arrEn[1] := bEn01;
arrEn[2] := bEn02;
arrEn[3] := bEn03;
arrEn[4] := bEn04;

arrVal[1] := bVal01;
arrVal[2] := bVal02;
arrVal[3] := bVal03;
arrVal[4] := bVal04;

bQ := FALSE;
bVal := FALSE;
nActvPrio := Const.nNoActvPrio;

FOR i := 1 TO cBA_PrioSwiB04 BY 1 DO
	IF	arrEn[i] = TRUE
	THEN
		bQ := TRUE;
		bVal := arrVal[i];
		nActvPrio := i;
		EXIT;
	END_IF
END_FOR

END_FUNCTION_BLOCK

// TEST/TestPackage/TEMPLATES/HeatSupply/HeatingCircuit/FB_Bnet_H_HtgCir_Sp
FUNCTION_BLOCK FB_Bnet_H_HtgCir_Sp EXTENDS FB_BACnet_View
VAR_INPUT
	rWthT			: REAL;
	nOpMod		: UDINT;	// Betriebsart	// Operating mode 
END_VAR
VAR_INPUT CONSTANT PERSISTENT
	HeatingSetpointProtection : REAL := 5;
END_VAR
VAR_OUTPUT
	rVal			: REAL;	//Sollwert Heizkreis//Setpoint heating circuit	
END_VAR
VAR_INPUT CONSTANT
	Curve							:	FB_Bnet_Scale_04 := (
											iParent			:= THIS^);
										
	NightOffs						:	FB_BACnet_AV_Setp := (
											iParent 			:= THIS^,
											sObjectName			:= '\/SP01',
											sDescription		:= '\/Sollwert Nachtabsenkung',
											eUnit				:= E_BA_Unit.eTemperature_DegreesCelsius,
											fValue				:= 8.0);

	SpFlWT							:	FB_BACnet_AV_Disp := (
											iParent 			:= THIS^,
											sObjectName			:= '\/SWC01',
											sDescription		:= '\/Errechnete Vorlauftemperatur',
											eUnit				:= E_BA_Unit.eTemperature_DegreesCelsius);
END_VAR
VAR
	PrioSwi			:	FB_MMUX_R04;//Priorisierung des Sollwertes//Prioritization of the setpoint
END_VAR
VAR // added by the converter: edge detectors and wires of the graphical bodies
    _w1 : ANY;
END_VAR

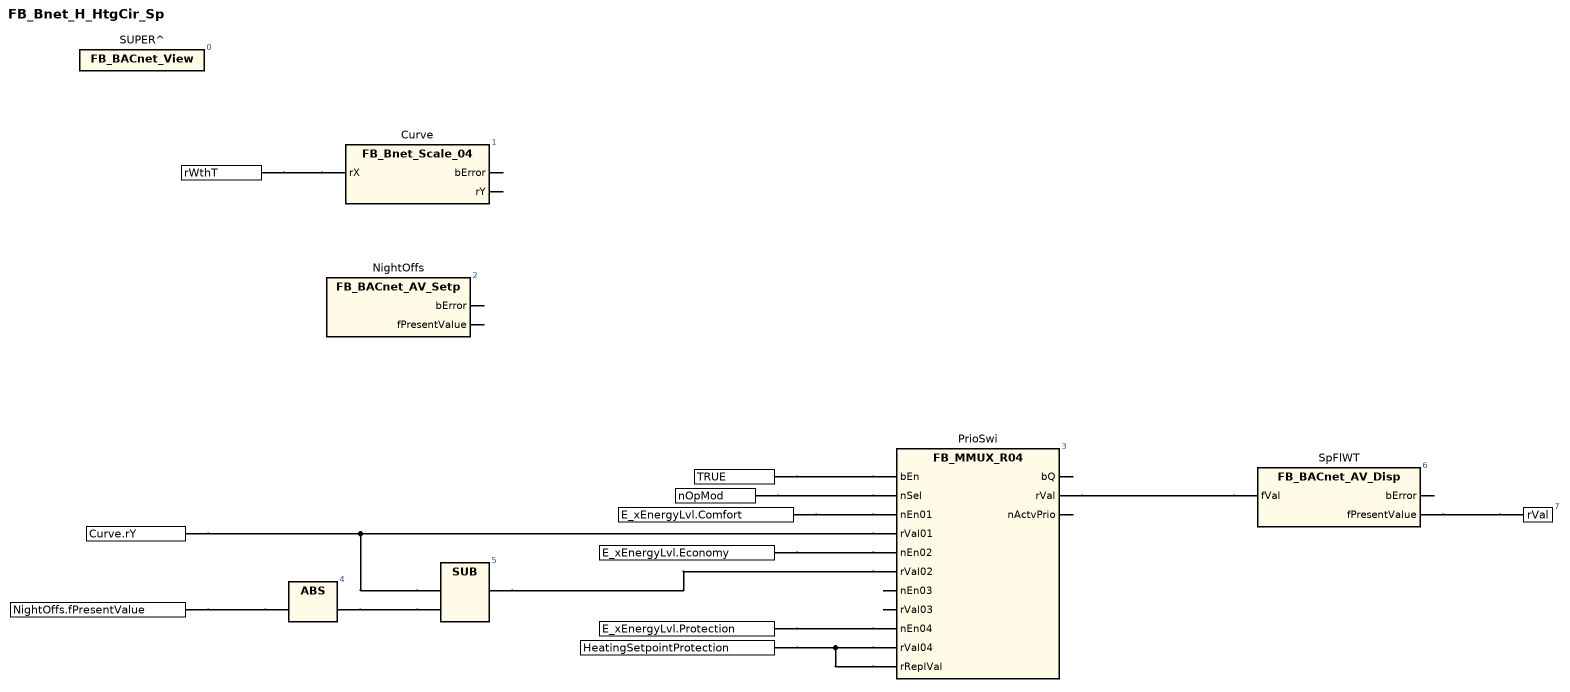
// note: 10 stored wires end on pins the file does not list and are not shown
SUPER^(); // FB_BACnet_View
Curve(rX := rWthT); // FB_Bnet_Scale_04
NightOffs(); // FB_BACnet_AV_Setp
PrioSwi(
    bEn := TRUE,
    nSel := nOpMod,
    nEn01 := E_xEnergyLvl.Comfort,
    rVal01 := Curve.rY,
    nEn02 := E_xEnergyLvl.Economy,
    rVal02 := _w1,
    nEn04 := E_xEnergyLvl.Protection,
    rVal04 := HeatingSetpointProtection,
    rReplVal := HeatingSetpointProtection); // FB_MMUX_R04
_w1 := Curve.rY - ABS(NightOffs.fPresentValue);
SpFlWT(fVal := PrioSwi.rVal); // FB_BACnet_AV_Disp
rVal := SpFlWT.fPresentValue;

METHOD FB_init : BOOL
VAR_INPUT
	bInitRetains : BOOL; // if TRUE, the retain variables are initialized (warm start / cold start)
	bInCopyCode : BOOL;  // if TRUE, the instance afterwards gets moved into the copy code (online change)
END_VAR
sObjectName		:= '\/SP01';
sDescription	:= '\/Sollwerte';
END_METHOD

END_FUNCTION_BLOCK

// TEST/TestPackage/TEMPLATES/Universal/Control/Scale/FB_Bnet_Scale_04
FUNCTION_BLOCK FB_Bnet_Scale_04 EXTENDS FB_BACnet_View
VAR_INPUT
	rX			:	REAL;	//	Istwert	//	Actual value
END_VAR
VAR_OUTPUT
	rY			:	REAL;	//	Skalierter Wert	//	scaled value
END_VAR
VAR
//Skalierung mit 4 Stützpunkten//Scaling with 4 interpolation points

	X1								:	FB_BACnet_AV_Setp := (
											iParent 			:= THIS^,
											sObjectName			:= '\/STX01',
											sDescription		:= '\/Stützpunkt X1',
											eUnit				:= E_BA_Unit.eTemperature_DegreesCelsius,
											fValue				:= 15);
	X2								:	FB_BACnet_AV_Setp := (
											iParent 			:= THIS^,
											sObjectName			:= '\/STX02',
											sDescription		:= '\/Stützpunkt X2',
											eUnit				:= E_BA_Unit.eTemperature_DegreesCelsius,
											fValue				:= 5);
	X3								:	FB_BACnet_AV_Setp := (
											iParent 			:= THIS^,
											sObjectName			:= '\/STX03',
											sDescription		:= '\/Stützpunkt X3',
											eUnit				:= E_BA_Unit.eTemperature_DegreesCelsius,
											fValue				:= 0);
	X4								:	FB_BACnet_AV_Setp := (
											iParent 			:= THIS^,
											sObjectName			:= '\/STX04',
											sDescription		:= '\/Stützpunkt X4',
											eUnit				:= E_BA_Unit.eTemperature_DegreesCelsius,
											fValue				:= -15);
											
	Y1								:	FB_BACnet_AV_Setp := (
											iParent 			:= THIS^,
											sObjectName			:= '\/STY01',
											sDescription		:= '\/Stützpunkt Y1',
											eUnit				:= E_BA_Unit.eTemperature_DegreesCelsius,
											fValue				:= 21);
	Y2								:	FB_BACnet_AV_Setp := (
											iParent 			:= THIS^,
											sObjectName			:= '\/STY02',
											sDescription		:= '\/Stützpunkt Y2',
											eUnit				:= E_BA_Unit.eTemperature_DegreesCelsius,
											fValue				:= 35);
	Y3								:	FB_BACnet_AV_Setp := (
											iParent 			:= THIS^,
											sObjectName			:= '\/STY03',
											sDescription		:= '\/Stützpunkt Y3',
											eUnit				:= E_BA_Unit.eTemperature_DegreesCelsius,
											fValue				:= 45);
	Y4								:	FB_BACnet_AV_Setp := (
											iParent 			:= THIS^,
											sObjectName			:= '\/STY04',
											sDescription		:= '\/Stützpunkt Y4',
											eUnit				:= E_BA_Unit.eTemperature_DegreesCelsius,
											fValue				:= 65);


	Scale			: FB_Chrct04;//Skalierungsfunktion//scaling function
	
	CalcSp							:	FB_BACnet_AV_Disp := (
											iParent 			:= THIS^,
											sObjectName			:= '\/CSP01',
											sDescription		:= '\/Errechneter Sollwert',
											eUnit				:= E_BA_Unit.eTemperature_DegreesCelsius);
END_VAR

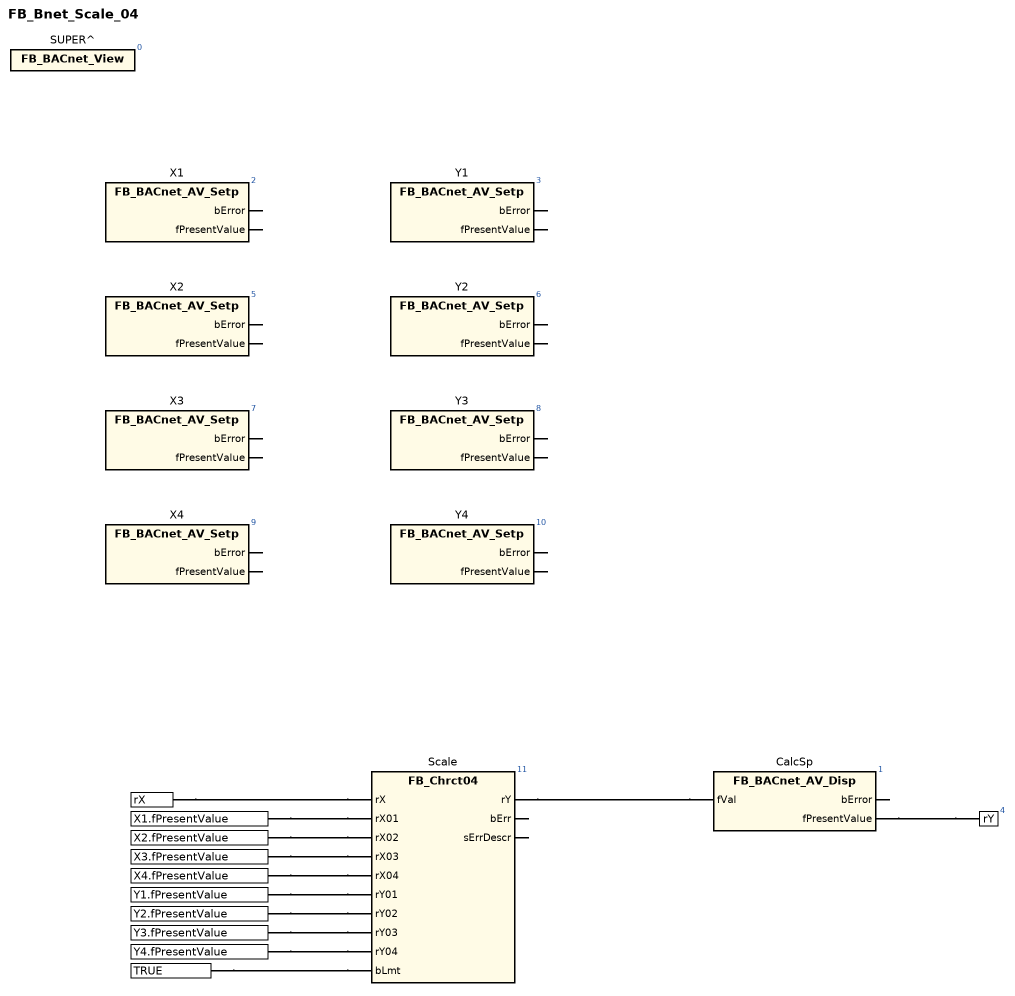
SUPER^(); // FB_BACnet_View
CalcSp(fVal := Scale.rY); // FB_BACnet_AV_Disp
X1(); // FB_BACnet_AV_Setp
Y1(); // FB_BACnet_AV_Setp
rY := CalcSp.fPresentValue;
X2(); // FB_BACnet_AV_Setp
Y2(); // FB_BACnet_AV_Setp
X3(); // FB_BACnet_AV_Setp
Y3(); // FB_BACnet_AV_Setp
X4(); // FB_BACnet_AV_Setp
Y4(); // FB_BACnet_AV_Setp
Scale(
    rX := rX,
    rX01 := X1.fPresentValue,
    rX02 := X2.fPresentValue,
    rX03 := X3.fPresentValue,
    rX04 := X4.fPresentValue,
    rY01 := Y1.fPresentValue,
    rY02 := Y2.fPresentValue,
    rY03 := Y3.fPresentValue,
    rY04 := Y4.fPresentValue,
    bLmt := TRUE); // FB_Chrct04

METHOD FB_init : BOOL
VAR_INPUT
	bInitRetains : BOOL; // if TRUE, the retain variables are initialized (warm start / cold start)
	bInCopyCode : BOOL;  // if TRUE, the instance afterwards gets moved into the copy code (online change)
END_VAR
sObjectName		:= '\/SCL01';
sDescription	:= '\/Kurve';
END_METHOD

END_FUNCTION_BLOCK

// TEST/TestPackage/TEMPLATES/Universal/Control/Scale/FB_Chrct04
FUNCTION_BLOCK FB_Chrct04
VAR_INPUT
	rX			: REAL;	// Input value of the characteristic curve
	rX01		: REAL;	// X-value for interpolation point P1
	rX02		: REAL;	// X-value for interpolation point P2
	rX03		: REAL;	// X-value for interpolation point P3
	rX04		: REAL;	// X-value for interpolation point P4
	rY01		: REAL;	// Y-value for interpolation point P1
	rY02		: REAL;	// Y-value for interpolation point P2
	rY03		: REAL;	// Y-value for interpolation point P3
	rY04		: REAL;	// Y-value for interpolation point P4	
	bLmt		: BOOL;		// True = Limitation lrY in range between Y1 and Y4
END_VAR
VAR_OUTPUT
	rY			: REAL;		// Calculated output value of the characteristic curve
	bErr		: BOOL;			// error
	sErrDescr	: T_MaxString;	// error description
END_VAR
VAR
	arrX			: ARRAY [1..cBA_NumOfElem] OF REAL;
	arrY			: ARRAY [1..cBA_NumOfElem] OF REAL;
	i				: UDINT;
	rM				: REAL;
	rBuffer1		: REAL;
	rBuffer2		: REAL;
END_VAR

VAR CONSTANT
	cBA_NumOfElem	: UDINT := 4;
END_VAR

	bErr     	:= FALSE;
	sErrDescr	:= '';

	arrX[1] := rX01;
	arrX[2] := rX02;
	arrX[3] := rX03;
	arrX[4] := rX04;
	
	arrY[1] := rY01;
	arrY[2] := rY02;
	arrY[3] := rY03;
	arrY[4] := rY04;

	FOR i := 1 TO (cBA_NumOfElem - 1) BY 1 DO
		rBuffer1 := arrX[i] - arrX[i + 1];
		rBuffer2 := 0;
		IF	MEMCMP(pBuf1 := ADR(rBuffer1), pBuf2 := ADR(rBuffer2), n := SIZEOF(rBuffer2)) = 0	THEN
			bErr		:= TRUE;
			sErrDescr	:= '01: Error at entered element no.';
			sErrDescr	:= CONCAT(sErrDescr, TO_STRING(i));
			sErrDescr	:= CONCAT(sErrDescr, '. The following sequence must be adhered to: lrX01 > lrX02 > lrXn OR lrX01 < lrX02 < lrXn');
			rY := 0;
			RETURN;
		END_IF
	END_FOR

(*Berechnung*)
(*X = (Y - Y1) / m + X1*)
	FOR i := 1 TO (cBA_NumOfElem - 1) BY 1 DO
		IF	rX >= arrX[i] AND rX <= arrX[i + 1] OR rX >= arrX[i + 1] AND rX <= arrX[i]	THEN
			(*lrM = Steigung*)
			(*m = (Y2 - Y1) / (X2 - X1*)
			rM := (arrY[i + 1] - arrY[i]) / (arrX[i + 1] - arrX[i]);
			(*Y = Y1 + m * (X - X1)*)
			rY := arrY[i] + rM * (rX - arrX[i]);
			RETURN;
		END_IF
	END_FOR

(*Berechnung wenn lrX ausserhalb von arrX[1] oder arrX[cNumOfEntries] liegt*)
	IF	arrX[1] > arrX[2] AND arrX[1] < rX OR arrX[1] < arrX[2] AND arrX[1] > rX	THEN
		(*lrM = Steigung*)
		(*m = (Y2 - Y1) / (X2 - X1*)
		rM := (rY02 - rY01) / (rX02 - rX01);
		(*Y = Y1 + m * (X - X1)*)
		rY := rY01 + rM * (rX - rX01);
	ELSIF	arrX[3] > arrX[cBA_NumOfElem] AND arrX[cBA_NumOfElem] > rX OR arrX[3] < arrX[cBA_NumOfElem] AND arrX[cBA_NumOfElem] < rX	THEN
		(*lrM = Steigung*)
		(*m = (Y4 - Y3) / (X4 - X3*)
		rM := (rY04 - rY03) / (rX04 - rX03);
		(*Y = Y3 + m * (X - X3)*)
		rY := rY03 + rM * (rX - rX03);
	END_IF

(*Limitierung der Bereichsgrenzen*)
	IF	bLmt	THEN
		IF	arrX[1] > arrX[2] AND arrX[1] < rX OR arrX[1] < arrX[2] AND arrX[1] > rX	THEN
			rY := rY01;
		END_IF
	
		IF	arrX[3] > arrX[cBA_NumOfElem] AND arrX[cBA_NumOfElem] > rX OR arrX[3] < arrX[cBA_NumOfElem] AND arrX[cBA_NumOfElem] < rX	THEN
			rY := rY04;
		END_IF
	END_IF

END_FUNCTION_BLOCK

// TEST/TestPackage/TEMPLATES/HeatSupply/HeatingCircuit/FB_MMUX_R04
FUNCTION_BLOCK FB_MMUX_R04
VAR_INPUT
	bEn			: BOOL;	// Activation of the block function
	nSel		: UDINT;// Selector
	nEn01		: UDINT := Const.nNoActvPrio;	// Input selector condition
	rVal01		: REAL;	// Input Value to chose from
	nEn02		: UDINT := Const.nNoActvPrio;	// Input selector condition
	rVal02		: REAL;	// Input Value to chose from
	nEn03		: UDINT := Const.nNoActvPrio;	// Input selector condition
	rVal03		: REAL;	// Input Value to chose from
	nEn04		: UDINT := Const.nNoActvPrio;	// Input selector condition
	rVal04		: REAL;	// Input Value to chose from
	rReplVal	: REAL;	// Substitute value, if no input selector condition is active
END_VAR
VAR_OUTPUT
	bQ			: BOOL;	// TRUE, if the selector nSel matches an input selector condition diNoActvPrio
	rVal		: REAL;	// Value of the selected input selector condition
	nActvPrio  : UDINT;	// Indicates which input selector condition is active
END_VAR

nSel := LIMIT(0,nSel,4294967294);

nActvPrio := Const.nNoActvPrio;
rVal := 0;
bQ := FALSE;

IF	bEn
THEN
	IF	nSel = nEn01
	THEN
		bQ := TRUE;
		rVal := rVal01;
		nActvPrio := 1;
		RETURN;
	END_IF
	
	IF	nSel = nEn02
	THEN
		bQ := TRUE;
		rVal := rVal02;
		nActvPrio := 2;
		RETURN;
	END_IF
	
	IF	nSel = nEn03
	THEN
		bQ := TRUE;
		rVal := rVal03;
		nActvPrio := 3;
		RETURN;
	END_IF
	
	IF	nSel = nEn04
	THEN
		bQ := TRUE;
		rVal := rVal04;
		nActvPrio := 4;
		RETURN;
	END_IF

	rVal := rReplVal;
END_IF

END_FUNCTION_BLOCK

// TEST/TestPackage/TEMPLATES/Universal/Valve/FB_Bnet_Vlv_013
FUNCTION_BLOCK FB_Bnet_Vlv_013 EXTENDS FB_BACnet_View
VAR_INPUT
	bEnSfty			: BOOL;
	fValSfty		: REAL;
	bEnCrit			: BOOL;
	fValCrit		: REAL;
	fValPgm			: REAL;
END_VAR
VAR_OUTPUT
	fPresentValue	: REAL;
	bEvent			: BOOL;
END_VAR
VAR
	AO								: FB_BACnet_AO_IO5P := (
										iParent 				:= THIS^,
										sObjectName				:= '\/CMD01',
										sDescription			:= '\/Schaltbefehl',
										sDeviceType				:= 'Ventil',
										fResolution				:= 0.003051851,
										fScaleOffset			:= 0,
										eUnit					:= E_BA_Unit.eOther_Percent);
END_VAR

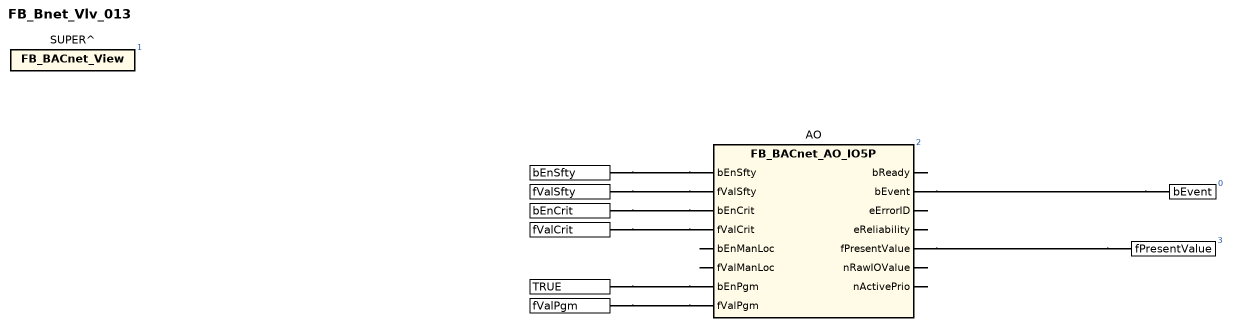
bEvent := AO.bEvent;
SUPER^(); // FB_BACnet_View
AO(
    bEnSfty := bEnSfty,
    fValSfty := fValSfty,
    bEnCrit := bEnCrit,
    fValCrit := fValCrit,
    bEnPgm := TRUE,
    fValPgm := fValPgm); // FB_BACnet_AO_IO5P
fPresentValue := AO.fPresentValue;

METHOD FB_init : BOOL
VAR_INPUT
	bInitRetains : BOOL; // if TRUE, the retain variables are initialized (warm start / cold start)
	bInCopyCode : BOOL;  // if TRUE, the instance afterwards gets moved into the copy code (online change)
END_VAR
sObjectName		:= '\/VLV01';
sDescription	:= '\/Ventil';
END_METHOD

END_FUNCTION_BLOCK

// TEST/TestPackage/TEMPLATES/Universal/Pump/1st/FB_Bnet_Pu1st
FUNCTION_BLOCK FB_Bnet_Pu1st EXTENDS FB_BACnet_View
VAR_INPUT
	bEnSfty		: BOOL;
	bValSfty	: BOOL;
	bEnCrit		: BOOL;
	bValCrit	: BOOL;
	bValPgm		: BOOL;
END_VAR
VAR_OUTPUT
	bQ			: BOOL;
END_VAR
VAR_INPUT CONSTANT
	Dst								: FB_BACnet_BI_IO := (
										iParent 				:= THIS^,
										sObjectName				:= '\/SM01',
										sDescription			:= '\/Störung',
										sDeviceType				:= 'Sicherung',
										sActiveText				:= 'Ausgelöst',
										sInactiveText			:= 'Normal',
										ePolarity				:= E_BA_Polarity.eReverse,
										nNotificationClass	:= 40,
										bEventEnable			:= [TRUE, TRUE, FALSE]);	
					
	BO								: FB_BACnet_BO_IO5P := (
										iParent 				:= THIS^,
										sObjectName				:= '\/CMD01',
										sDescription			:= '\/Schaltbefehl',
										sDeviceType				:= 'Ausgang',
										sActiveText				:= 'Ein',
										sInactiveText			:= 'Aus');

	DlyOff							: FB_Bnet_DlyOff := (
										iParent 				:= THIS^);

	Ablk							: FB_Bnet_AntiBlocking := (
										iParent 				:= THIS^);
END_VAR
VAR // added by the converter: edge detectors and wires of the graphical bodies
    _w1 : BOOL;
END_VAR

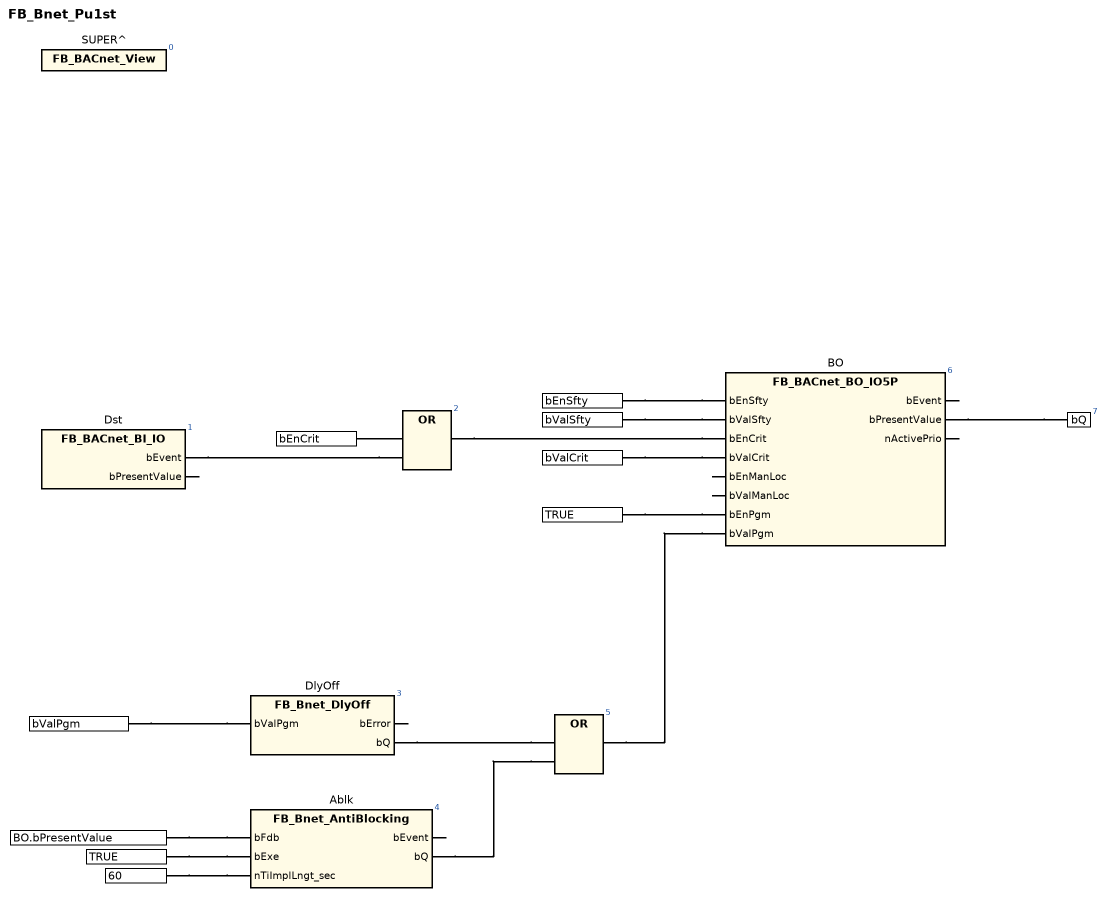
SUPER^(); // FB_BACnet_View
Dst(); // FB_BACnet_BI_IO
_w1 := bEnCrit OR Dst.bEvent;
DlyOff(bValPgm := bValPgm); // FB_Bnet_DlyOff
Ablk(bFdb := BO.bPresentValue, bExe := TRUE, nTiImplLngt_sec := 60); // FB_Bnet_AntiBlocking
BO(
    bEnSfty := bEnSfty,
    bValSfty := bValSfty,
    bEnCrit := _w1,
    bValCrit := bValCrit,
    bEnPgm := TRUE,
    bValPgm := DlyOff.bQ OR Ablk.bQ); // FB_BACnet_BO_IO5P
bQ := BO.bPresentValue;

METHOD FB_init : BOOL
VAR_INPUT
	bInitRetains : BOOL; // if TRUE, the retain variables are initialized (warm start / cold start)
	bInCopyCode : BOOL;  // if TRUE, the instance afterwards gets moved into the copy code (online change)
END_VAR
sObjectName		:= '\/PU01';
sDescription	:= '\/Pumpe';
END_METHOD

END_FUNCTION_BLOCK

// TEST/TestPackage/TEMPLATES/Universal/Control/DelayOff/FB_Bnet_DlyOff
FUNCTION_BLOCK FB_Bnet_DlyOff EXTENDS FB_BACnet_View
VAR_INPUT
	bValPgm		:	BOOL;	//	Wert Programmpriorität		//	Value program priority
END_VAR
VAR_OUTPUT
	bQ			:	BOOL;	//	aktiv	//	active
END_VAR
VAR
	TiVal							:	FB_BACnet_AV_Setp := (
											iParent 			:= THIS^,
											sObjectName			:= '\/SP01',
											sDescription		:= '\/Sollwert',
											eUnit				:= E_BA_Unit.eTime_Seconds,
											fValue				:= 0);
											
	tofDlyOff	: TOF; // Zeitglied Aktor verzögert aus	// Timer actuator delay off
END_VAR

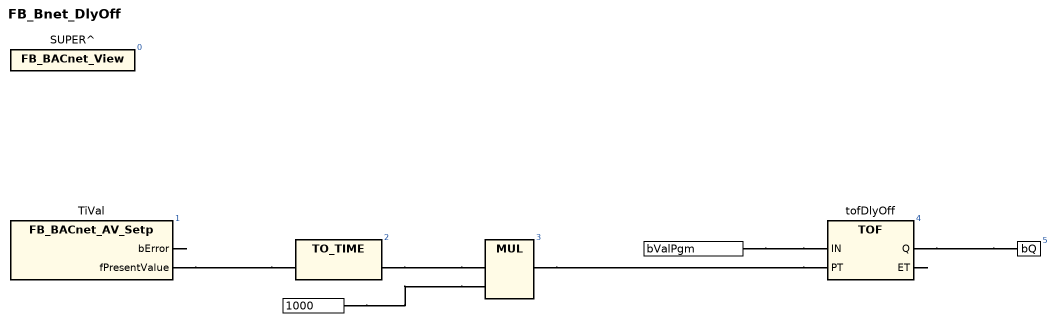
SUPER^(); // FB_BACnet_View
TiVal(); // FB_BACnet_AV_Setp
tofDlyOff(IN := bValPgm, PT := TO_TIME(TiVal.fPresentValue) * 1000); // TOF
bQ := tofDlyOff.Q;

METHOD FB_init : BOOL
VAR_INPUT
	bInitRetains : BOOL; // if TRUE, the retain variables are initialized (warm start / cold start)
	bInCopyCode : BOOL;  // if TRUE, the instance afterwards gets moved into the copy code (online change)
END_VAR
sObjectName		:= '\/DLY01';
sDescription	:= '\/Ausschaltverzögerung';
END_METHOD

END_FUNCTION_BLOCK

// TEST/TestPackage/TEMPLATES/Universal/AntiBlocking/FB_Bnet_AntiBlocking
FUNCTION_BLOCK FB_Bnet_AntiBlocking EXTENDS FB_BACnet_View
VAR_INPUT CONSTANT PERSISTENT
	bEn				:	BOOL := TRUE;
END_VAR
VAR_INPUT
	bFdb					:	BOOL;	
	bExe					:	BOOL;
	nTiImplLngt_sec			:	UDINT;
END_VAR
VAR_OUTPUT
	bQ			:	BOOL;	//	aktiv	//	active
END_VAR
VAR
	IdlePrd							:	FB_BACnet_AV_Setp := (
											iParent 			:= THIS^,
											sObjectName			:= '\/SP01',
											sDescription		:= '\/Sollwert',
											eUnit				:= E_BA_Unit.eTime_Hours,
											fValue				:= 168);
											
	AblkFnct		: FB_AntBlkg; // Antiblockierschutzfunktion Pumpe	// anti-blocking protection function pump
END_VAR

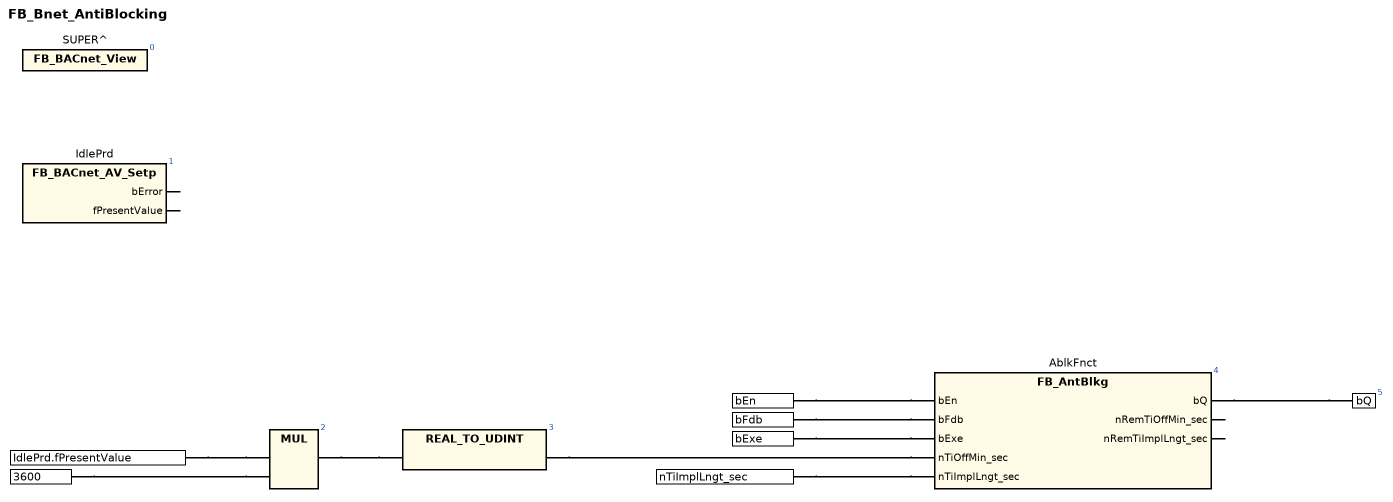
SUPER^(); // FB_BACnet_View
IdlePrd(); // FB_BACnet_AV_Setp
AblkFnct(
    bEn := bEn,
    bFdb := bFdb,
    bExe := bExe,
    nTiOffMin_sec := REAL_TO_UDINT(IdlePrd.fPresentValue * 3600),
    nTiImplLngt_sec := nTiImplLngt_sec); // FB_AntBlkg
bQ := AblkFnct.bQ;

METHOD FB_init : BOOL
VAR_INPUT
	bInitRetains : BOOL; // if TRUE, the retain variables are initialized (warm start / cold start)
	bInCopyCode : BOOL;  // if TRUE, the instance afterwards gets moved into the copy code (online change)
END_VAR
sObjectName		:= '\/RZ01';
sDescription	:= '\/Blockierschutz';
END_METHOD

END_FUNCTION_BLOCK

// TEST/TestPackage/TEMPLATES/Universal/AntiBlocking/FB_AntBlkg
FUNCTION_BLOCK FB_AntBlkg
VAR_INPUT
	bEn					: BOOL;// enables the function block
	bFdb				: BOOL;// input for connecting the feedback signal of a motor or valve
	bExe				: BOOL;// rising edge forces a pulse output
	nTiOffMin_sec		: UDINT;// (0..Const.nTiSec) minimum switch-off time [s]: A pulse is issued once the time nTiOffMin has elapsed without movement of the unit
	nTiImplLngt_sec		: UDINT;// (0..Const.nTiSec) length of the blocking protection pulse [s] at bQ
END_VAR
VAR_OUTPUT
	bQ                  : BOOL;// pulse output
	nRemTiOffMin_sec    : UDINT;// remaining time [s] before the next pulse is issued in the absence of movement
	nRemTiImplLngt_sec  : UDINT;// remaining residual time [s] of the pulse at bQ
END_VAR
VAR
	tonTiOffMin			: TON;
	tTiOffMin			: TIME;
	tonImplLngt			: TON;
	tImplLngt			: TIME;
	nStep				: INT;
END_VAR

(*============================*)
tTiOffMin := TO_TIME(1000 * nTiOffMin_sec);
tImplLngt := TO_TIME(1000 * nTiImplLngt_sec);
(*============================*)

CASE nStep OF
0:
	nRemTiImplLngt_sec := 0;
	bQ := FALSE;
	tonImplLngt(IN := FALSE, PT := T#0s);
	tonTiOffMin(IN := bEn AND NOT bFdb, PT := tTiOffMin);
	nRemTiOffMin_sec := F_RemSecsTon(tonTimer := tonTiOffMin);

	IF	tonTiOffMin.Q AND bExe
	THEN
		bQ := TRUE;
		nStep := 10;
	END_IF

10:
	nRemTiOffMin_sec := 0;
	tonTiOffMin(IN := FALSE, PT := T#0s);
	tonImplLngt(IN := TRUE, PT := tImplLngt);
	nRemTiImplLngt_sec := F_RemSecsTon(tonTimer := tonImplLngt);

	IF	tonImplLngt.Q OR
		NOT bEn
	THEN
		nStep := 0;
	END_IF
END_CASE

END_FUNCTION_BLOCK

// TEST/TestPackage/Structure Samples/PRG02/TEMPLATES/Custom/H/HtgCirABC123/FB_BA_HtgCirABC123_Vlv
FUNCTION_BLOCK FB_BA_HtgCirABC123_Vlv EXTENDS FB_BACnet_View
VAR_INPUT
	bEnSfty			: BOOL;
	fValSfty		: REAL;
	bEnCrit			: BOOL;
	fValCrit		: REAL;
	fValPgm			: REAL;
END_VAR
VAR_OUTPUT
	fPresentValue	: REAL;
	bEvent			: BOOL;
END_VAR
VAR
	AO								: FB_BACnet_AO_IO5P := (
										iParent 				:= THIS^,
										sObjectName				:= '\/CMD01',
										sDescription			:= '\/Schaltbefehl',
										sDeviceType				:= 'Ventil',
										fResolution				:= 0.003051851,
										fScaleOffset			:= 0,
										eUnit					:= E_BA_Unit.eOther_Percent);
END_VAR

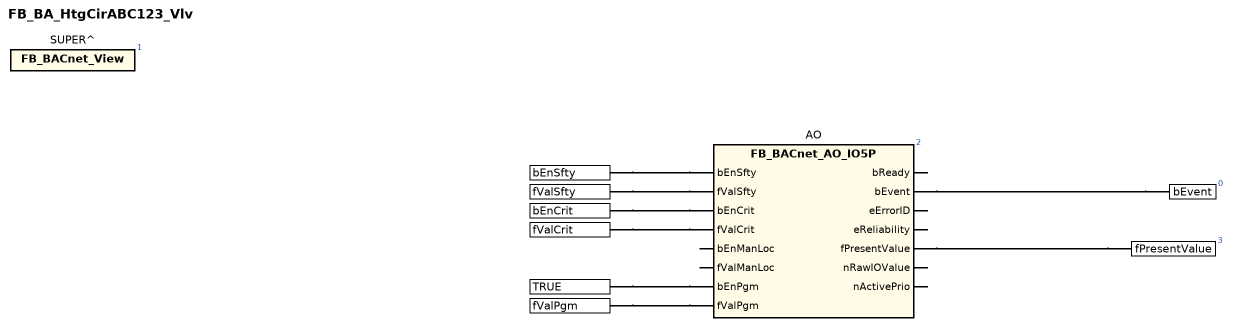
bEvent := AO.bEvent;
SUPER^(); // FB_BACnet_View
AO(
    bEnSfty := bEnSfty,
    fValSfty := fValSfty,
    bEnCrit := bEnCrit,
    fValCrit := fValCrit,
    bEnPgm := TRUE,
    fValPgm := fValPgm); // FB_BACnet_AO_IO5P
fPresentValue := AO.fPresentValue;

METHOD FB_init : BOOL
VAR_INPUT
	bInitRetains : BOOL; // if TRUE, the retain variables are initialized (warm start / cold start)
	bInCopyCode : BOOL;  // if TRUE, the instance afterwards gets moved into the copy code (online change)
END_VAR
sObjectName		:= '\/VLV01';
sDescription	:= '\/Ventil';
END_METHOD

END_FUNCTION_BLOCK

// TEST/TestPackage/Structure Samples/PRG02/TEMPLATES/Custom/H/HtgCirTZU555/FB_BA_HtgCirTZU555
FUNCTION_BLOCK FB_BA_HtgCirTZU555 EXTENDS FB_BACnet_View
VAR_INPUT CONSTANT
	WthT							: FB_BACnet_AI_IO := (
										iParent 					:= THIS^,
										sObjectName					:= '\/WTHT',
										sDescription				:= '\/Aussentemperatur',
										sDeviceType					:= 'Temperatursensor',
										fResolution					:= 0.003051851,
										eUnit						:= E_BA_Unit.eTemperature_DegreesCelsius);
										
	FlWT							: FB_BACnet_AI_IO := (
										iParent 					:= THIS^,
										sObjectName					:= '\/TVL',
										sDescription				:= '\/Vorlauftemperatur',
										sDeviceType					:= 'Temperatursensor',
										fResolution					:= 0.003051851,
										eUnit						:= E_BA_Unit.eTemperature_DegreesCelsius);
	RtWT							: FB_BACnet_AI_IO := (
										iParent 					:= THIS^,
										sObjectName					:= '\/TRT',
										sDescription				:= '\/Rücklauftemperatur',
										sDeviceType					:= 'Temperatursensor',
										fResolution					:= 0.003051851,
										fScaleOffset				:= 0,
										eUnit						:= E_BA_Unit.eTemperature_DegreesCelsius);
										
	Sched							: FB_BACnet_SchedB := (
										iParent 					:= THIS^,
										sObjectName					:= '\/SCH01',
										sDescription				:= '\/Zeitschaltprogramm',
										tWeek						:= F_BACnet_SchedWeekly3xB(E_BA_Weekday.eMonday, E_BA_Weekday.eFriday, T#0H, FALSE, T#6H, TRUE, T#20H, FALSE));
										
	PID								: FB_BACnet_Loop := (
										iParent 					:= THIS^,
										sObjectName					:= '\/PID01',
										sDescription				:= '\/Vorlauftemperatirregler',
										eAction						:= E_BA_Action.eReverse,
										fPropertionalConstant		:= 1,
										fIntegralConstant			:= 180);	
										
	OpM								: FB_Bnet_H_OpM := (
										iParent 					:= THIS^);	
										
	SpG								: FB_Bnet_H_HtgCir_Sp := (
										iParent 					:= THIS^);	
										
	HtgLimit						: FB_Bnet_H_HtgCir_HtgLmt := (
										iParent 					:= THIS^);
										
	Vlv								: FB_Bnet_Vlv_013 := (
										iParent 					:= THIS^);	
										
	Pu								: FB_Bnet_Pu1st := (
										iParent 					:= THIS^);	
END_VAR
VAR // added by the converter: edge detectors and wires of the graphical bodies
    _w1 : ANY;
END_VAR

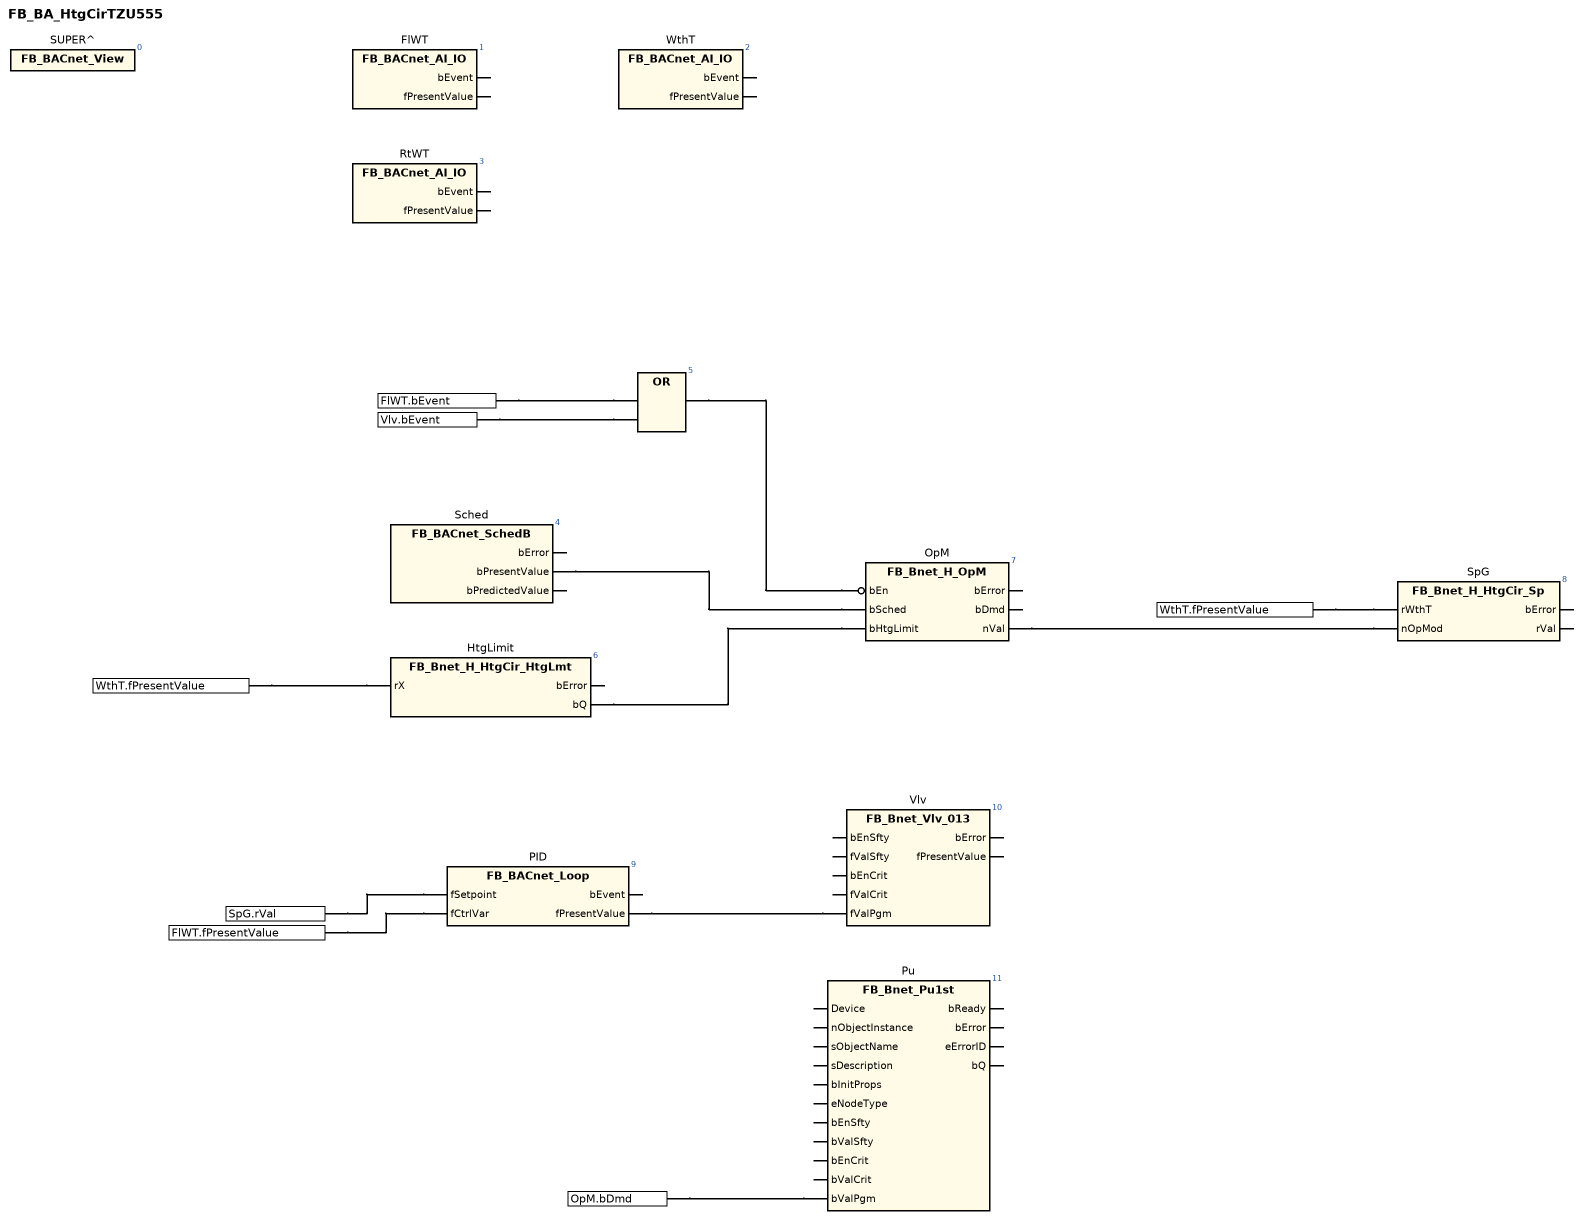
// note: 28 stored wires end on pins the file does not list and are not shown
SUPER^(); // FB_BACnet_View
FlWT(); // FB_BACnet_AI_IO
WthT(); // FB_BACnet_AI_IO
RtWT(); // FB_BACnet_AI_IO
Sched(); // FB_BACnet_SchedB
_w1 := FlWT.bEvent OR Vlv.bEvent;
HtgLimit(rX := WthT.fPresentValue); // FB_Bnet_H_HtgCir_HtgLmt
OpM(bEn := NOT _w1, bSched := Sched.bPresentValue, bHtgLimit := HtgLimit.bQ); // FB_Bnet_H_OpM
SpG(rWthT := WthT.fPresentValue, nOpMod := OpM.nVal); // FB_Bnet_H_HtgCir_Sp
PID(fSetpoint := SpG.rVal, fCtrlVar := FlWT.fPresentValue); // FB_BACnet_Loop
Vlv(fValPgm := PID.fPresentValue); // FB_Bnet_Vlv_013
Pu(bValPgm := OpM.bDmd); // FB_Bnet_Pu1st

METHOD FB_init : BOOL
VAR_INPUT
	bInitRetains : BOOL; // if TRUE, the retain variables are initialized (warm start / cold start)
	bInCopyCode : BOOL;  // if TRUE, the instance afterwards gets moved into the copy code (online change)
END_VAR
sObjectName		:= '\/HCR01';
sDescription	:= '\/Heizkreis';

Pu.BO.sObjectName := '\/XXXtest';
END_METHOD

END_FUNCTION_BLOCK

// TEST/TestPackage/Structure Samples/PRG02/TEMPLATES/Custom/H/HtgCirTZU555/FB_BA_HtgCirTZU555_Pu
FUNCTION_BLOCK FB_BA_HtgCirTZU555_Pu EXTENDS FB_BACnet_View
VAR_INPUT
	bEnSfty			: BOOL;
	fValSfty		: REAL;
	bEnCrit			: BOOL;
	fValCrit		: REAL;
	fValPgm			: REAL;
END_VAR
VAR_OUTPUT
	fPresentValue	: REAL;
	bEvent			: BOOL;
END_VAR
VAR
	AO								: FB_BACnet_AO_IO5P := (
										iParent 				:= THIS^,
										sObjectName				:= '\/CMD01',
										sDescription			:= '\/Schaltbefehl',
										sDeviceType				:= 'Ventil',
										fResolution				:= 0.003051851,
										fScaleOffset			:= 0,
										eUnit					:= E_BA_Unit.eOther_Percent);
END_VAR

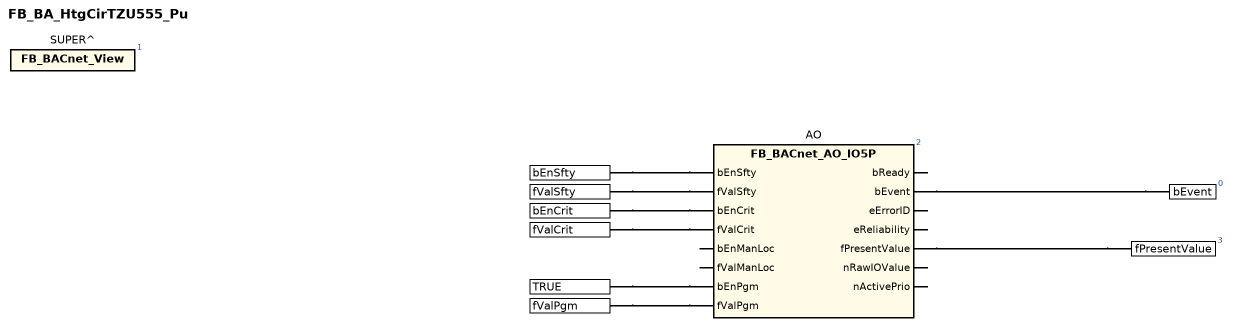
bEvent := AO.bEvent;
SUPER^(); // FB_BACnet_View
AO(
    bEnSfty := bEnSfty,
    fValSfty := fValSfty,
    bEnCrit := bEnCrit,
    fValCrit := fValCrit,
    bEnPgm := TRUE,
    fValPgm := fValPgm); // FB_BACnet_AO_IO5P
fPresentValue := AO.fPresentValue;

METHOD FB_init : BOOL
VAR_INPUT
	bInitRetains : BOOL; // if TRUE, the retain variables are initialized (warm start / cold start)
	bInCopyCode : BOOL;  // if TRUE, the instance afterwards gets moved into the copy code (online change)
END_VAR
sObjectName		:= '\/VLV01';
sDescription	:= '\/Ventil';
END_METHOD

END_FUNCTION_BLOCK

// TEST/TestPackage/Structure Samples/PRG02/TEMPLATES/Standard/AC/FB_BA_AC01
FUNCTION_BLOCK FB_BA_AC01 EXTENDS FB_BACnet_View
VAR_INPUT CONSTANT
	WthT							: FB_BACnet_AI_IO := (
										iParent 					:= THIS^,
										sObjectName					:= '\/WTHT',
										sDescription				:= '\/Aussentemperatur',
										sDeviceType					:= 'Temperatursensor',
										fResolution					:= 0.003051851,
										eUnit						:= E_BA_Unit.eTemperature_DegreesCelsius);
										
	FlWT							: FB_BACnet_AI_IO := (
										iParent 					:= THIS^,
										sObjectName					:= '\/TVL',
										sDescription				:= '\/Vorlauftemperatur',
										sDeviceType					:= 'Temperatursensor',
										fResolution					:= 0.003051851,
										eUnit						:= E_BA_Unit.eTemperature_DegreesCelsius);
	RtWT							: FB_BACnet_AI_IO := (
										iParent 					:= THIS^,
										sObjectName					:= '\/TRT',
										sDescription				:= '\/Rücklauftemperatur',
										sDeviceType					:= 'Temperatursensor',
										fResolution					:= 0.003051851,
										fScaleOffset				:= 0,
										eUnit						:= E_BA_Unit.eTemperature_DegreesCelsius);
										
	Sched							: FB_BACnet_SchedB := (
										iParent 					:= THIS^,
										sObjectName					:= '\/SCH01',
										sDescription				:= '\/Zeitschaltprogramm',
										tWeek						:= F_BACnet_SchedWeekly3xB(E_BA_Weekday.eMonday, E_BA_Weekday.eFriday, T#0H, FALSE, T#6H, TRUE, T#20H, FALSE));
										
	PID								: FB_BACnet_Loop := (
										iParent 					:= THIS^,
										sObjectName					:= '\/PID01',
										sDescription				:= '\/Vorlauftemperatirregler',
										eAction						:= E_BA_Action.eReverse,
										fPropertionalConstant		:= 1,
										fIntegralConstant			:= 180);	
										
	OpM								: FB_Bnet_H_OpM := (
										iParent 					:= THIS^);	
										
	SpG								: FB_Bnet_H_HtgCir_Sp := (
										iParent 					:= THIS^);	
										
	HtgLimit						: FB_Bnet_H_HtgCir_HtgLmt := (
										iParent 					:= THIS^);
										
	Vlv								: FB_Bnet_Vlv_013 := (
										iParent 					:= THIS^);	
										
	Pu								: FB_Bnet_Pu1st := (
										iParent 					:= THIS^);	
END_VAR
VAR // added by the converter: edge detectors and wires of the graphical bodies
    _w1 : ANY;
END_VAR

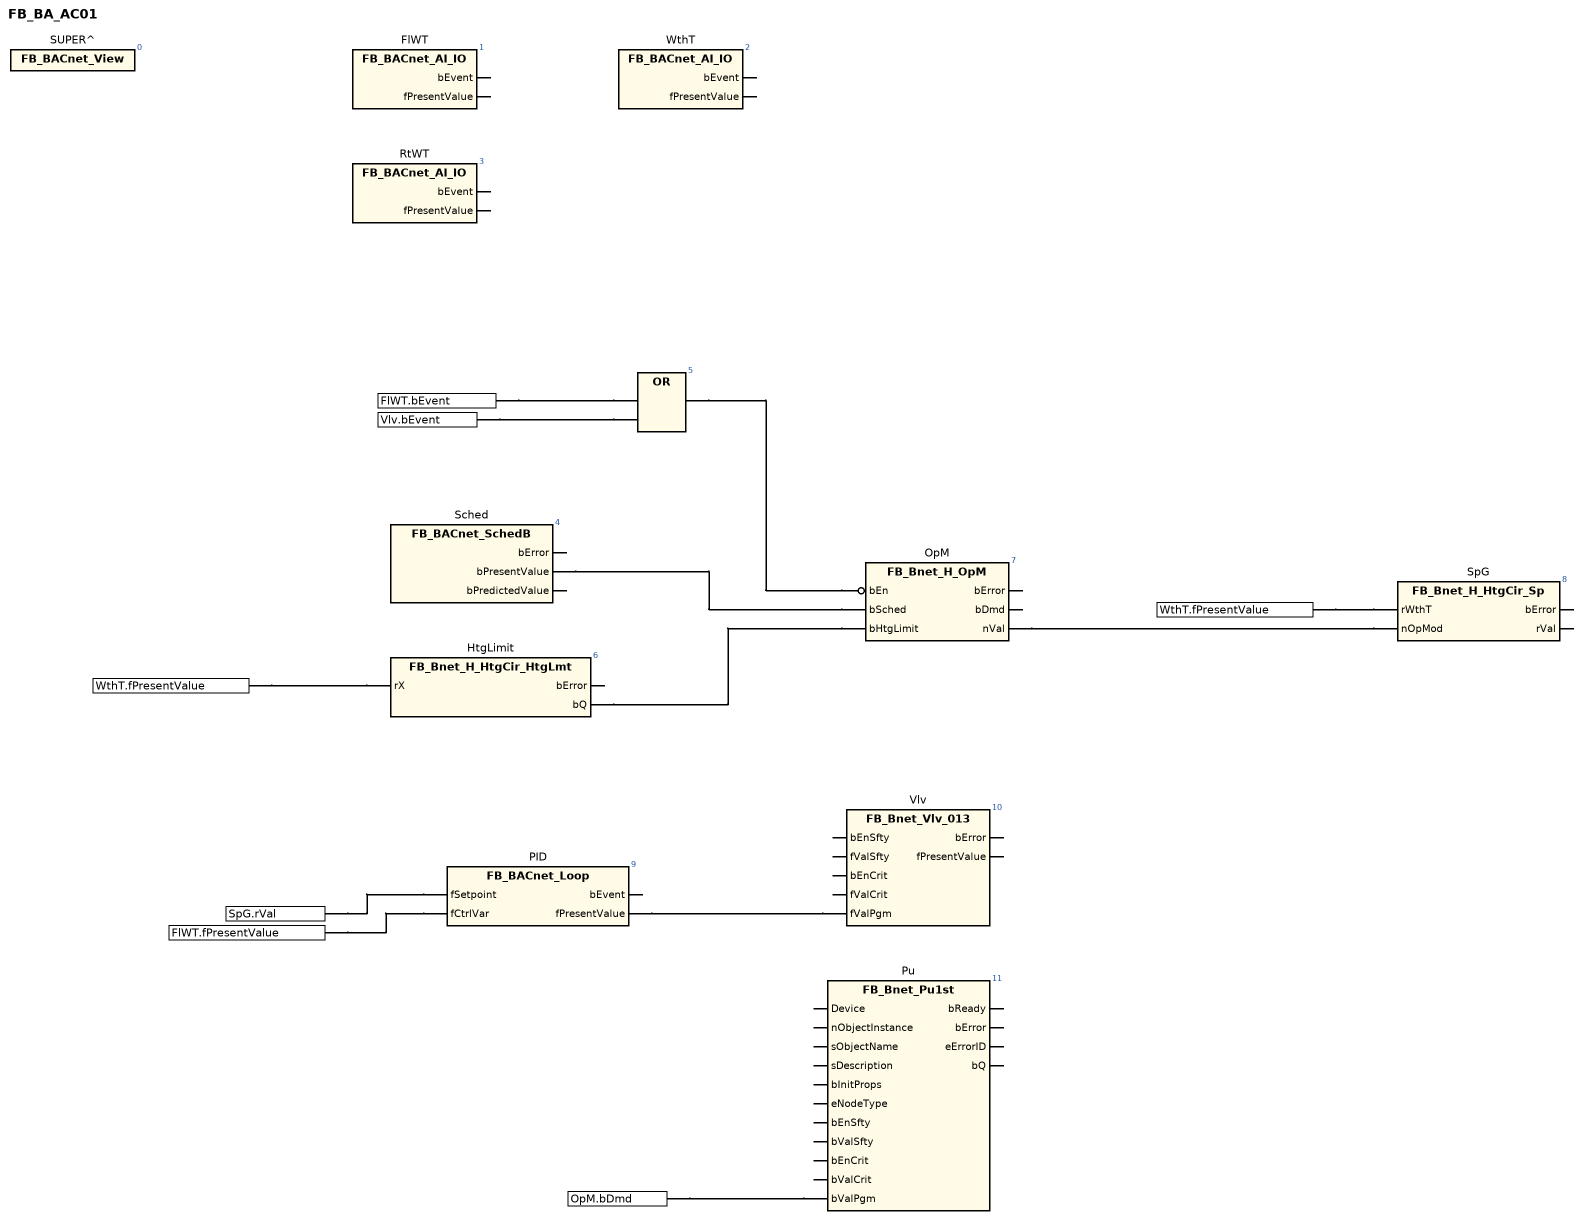
// note: 28 stored wires end on pins the file does not list and are not shown
SUPER^(); // FB_BACnet_View
FlWT(); // FB_BACnet_AI_IO
WthT(); // FB_BACnet_AI_IO
RtWT(); // FB_BACnet_AI_IO
Sched(); // FB_BACnet_SchedB
_w1 := FlWT.bEvent OR Vlv.bEvent;
HtgLimit(rX := WthT.fPresentValue); // FB_Bnet_H_HtgCir_HtgLmt
OpM(bEn := NOT _w1, bSched := Sched.bPresentValue, bHtgLimit := HtgLimit.bQ); // FB_Bnet_H_OpM
SpG(rWthT := WthT.fPresentValue, nOpMod := OpM.nVal); // FB_Bnet_H_HtgCir_Sp
PID(fSetpoint := SpG.rVal, fCtrlVar := FlWT.fPresentValue); // FB_BACnet_Loop
Vlv(fValPgm := PID.fPresentValue); // FB_Bnet_Vlv_013
Pu(bValPgm := OpM.bDmd); // FB_Bnet_Pu1st

METHOD FB_init : BOOL
VAR_INPUT
	bInitRetains : BOOL; // if TRUE, the retain variables are initialized (warm start / cold start)
	bInCopyCode : BOOL;  // if TRUE, the instance afterwards gets moved into the copy code (online change)
END_VAR
sObjectName		:= '\/HCR01';
sDescription	:= '\/Heizkreis';

Pu.BO.sObjectName := '\/XXXtest';
END_METHOD

END_FUNCTION_BLOCK

// TEST/TestPackage/Structure Samples/PRG02/TEMPLATES/Standard/H/FB_BA_HtgCir01
FUNCTION_BLOCK FB_BA_HtgCir01 EXTENDS FB_BACnet_View
VAR_INPUT CONSTANT
	WthT							: FB_BACnet_AI_IO := (
										iParent 					:= THIS^,
										sObjectName					:= '\/WTHT',
										sDescription				:= '\/Aussentemperatur',
										sDeviceType					:= 'Temperatursensor',
										fResolution					:= 0.003051851,
										eUnit						:= E_BA_Unit.eTemperature_DegreesCelsius);
										
	FlWT							: FB_BACnet_AI_IO := (
										iParent 					:= THIS^,
										sObjectName					:= '\/TVL',
										sDescription				:= '\/Vorlauftemperatur',
										sDeviceType					:= 'Temperatursensor',
										fResolution					:= 0.003051851,
										eUnit						:= E_BA_Unit.eTemperature_DegreesCelsius);
	RtWT							: FB_BACnet_AI_IO := (
										iParent 					:= THIS^,
										sObjectName					:= '\/TRT',
										sDescription				:= '\/Rücklauftemperatur',
										sDeviceType					:= 'Temperatursensor',
										fResolution					:= 0.003051851,
										fScaleOffset				:= 0,
										eUnit						:= E_BA_Unit.eTemperature_DegreesCelsius);
										
	Sched							: FB_BACnet_SchedB := (
										iParent 					:= THIS^,
										sObjectName					:= '\/SCH01',
										sDescription				:= '\/Zeitschaltprogramm',
										tWeek						:= F_BACnet_SchedWeekly3xB(E_BA_Weekday.eMonday, E_BA_Weekday.eFriday, T#0H, FALSE, T#6H, TRUE, T#20H, FALSE));
										
	PID								: FB_BACnet_Loop := (
										iParent 					:= THIS^,
										sObjectName					:= '\/PID01',
										sDescription				:= '\/Vorlauftemperatirregler',
										eAction						:= E_BA_Action.eReverse,
										fPropertionalConstant		:= 1,
										fIntegralConstant			:= 180);	
										
	OpM								: FB_Bnet_H_OpM := (
										iParent 					:= THIS^);	
										
	SpG								: FB_Bnet_H_HtgCir_Sp := (
										iParent 					:= THIS^);	
										
	HtgLimit						: FB_Bnet_H_HtgCir_HtgLmt := (
										iParent 					:= THIS^);
										
	Vlv								: FB_Bnet_Vlv_013 := (
										iParent 					:= THIS^);	
										
	Pu								: FB_Bnet_Pu1st := (
										iParent 					:= THIS^);	
END_VAR
VAR // added by the converter: edge detectors and wires of the graphical bodies
    _w1 : ANY;
END_VAR

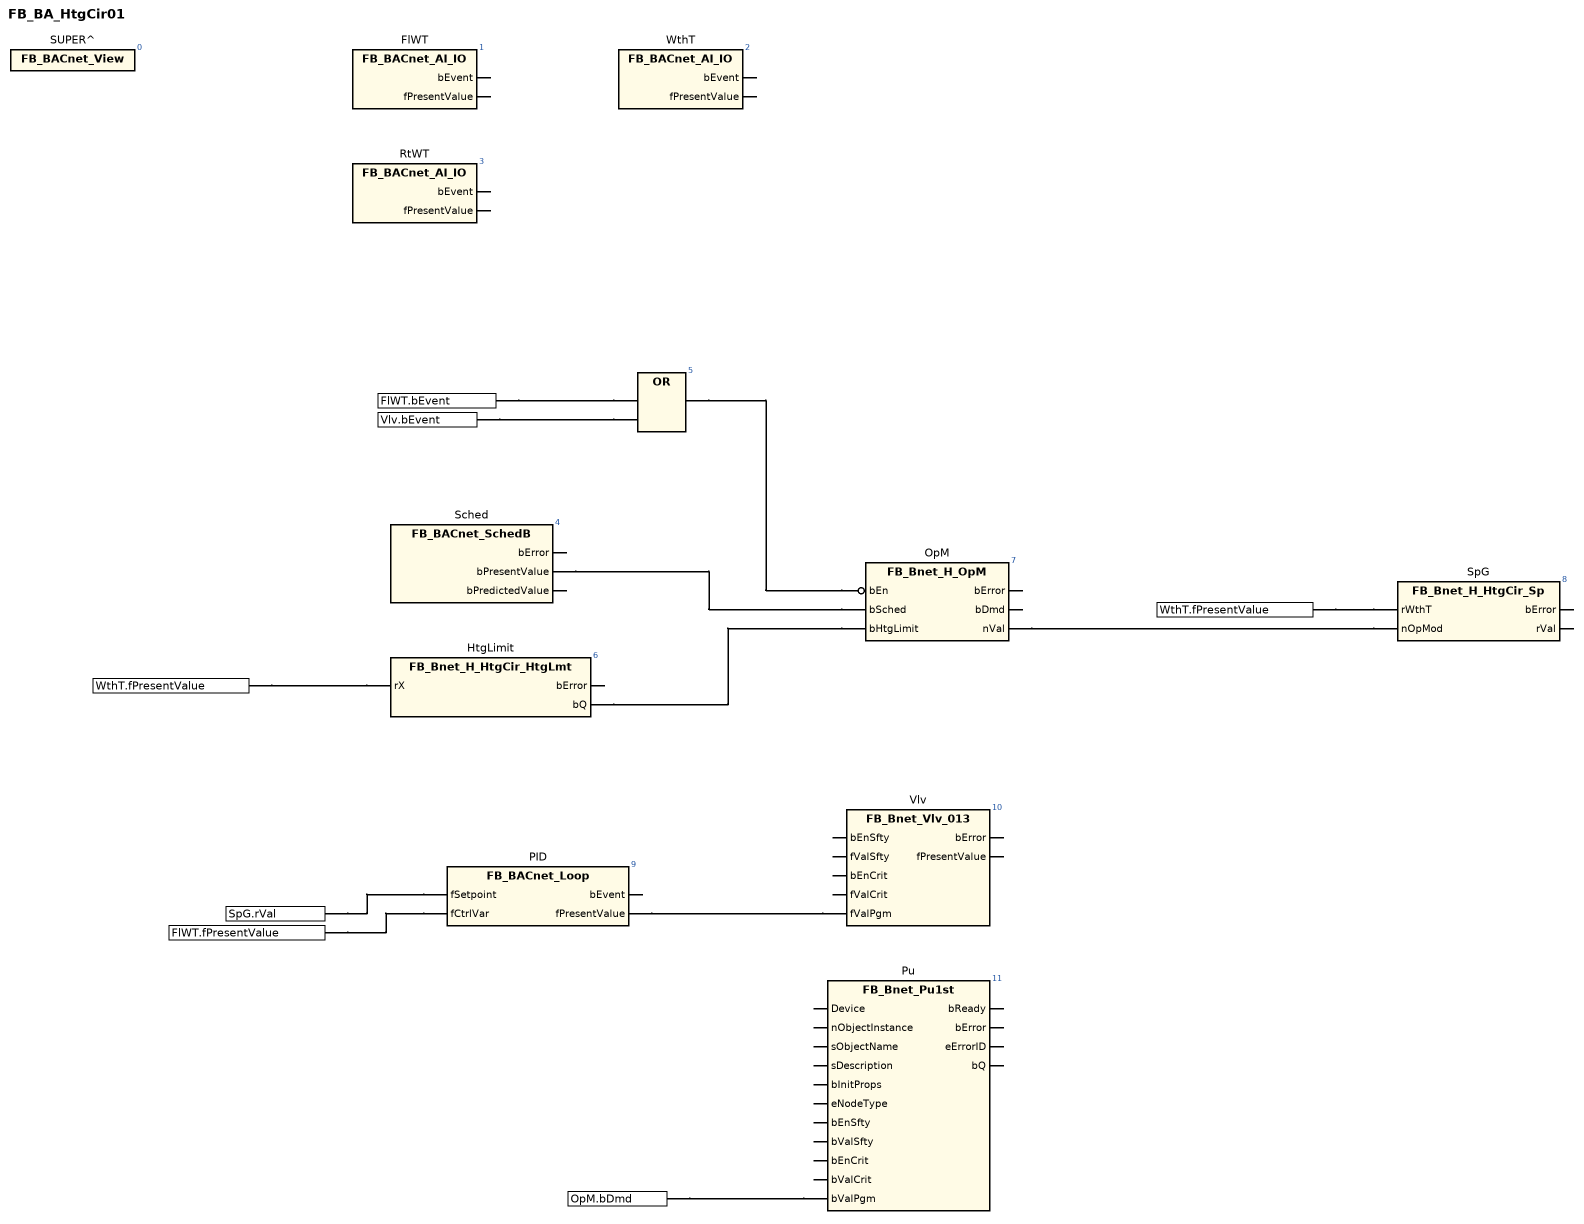
// note: 28 stored wires end on pins the file does not list and are not shown
SUPER^(); // FB_BACnet_View
FlWT(); // FB_BACnet_AI_IO
WthT(); // FB_BACnet_AI_IO
RtWT(); // FB_BACnet_AI_IO
Sched(); // FB_BACnet_SchedB
_w1 := FlWT.bEvent OR Vlv.bEvent;
HtgLimit(rX := WthT.fPresentValue); // FB_Bnet_H_HtgCir_HtgLmt
OpM(bEn := NOT _w1, bSched := Sched.bPresentValue, bHtgLimit := HtgLimit.bQ); // FB_Bnet_H_OpM
SpG(rWthT := WthT.fPresentValue, nOpMod := OpM.nVal); // FB_Bnet_H_HtgCir_Sp
PID(fSetpoint := SpG.rVal, fCtrlVar := FlWT.fPresentValue); // FB_BACnet_Loop
Vlv(fValPgm := PID.fPresentValue); // FB_Bnet_Vlv_013
Pu(bValPgm := OpM.bDmd); // FB_Bnet_Pu1st

METHOD FB_init : BOOL
VAR_INPUT
	bInitRetains : BOOL; // if TRUE, the retain variables are initialized (warm start / cold start)
	bInCopyCode : BOOL;  // if TRUE, the instance afterwards gets moved into the copy code (online change)
END_VAR
sObjectName		:= '\/HCR01';
sDescription	:= '\/Heizkreis';

Pu.BO.sObjectName := '\/XXXtest';
END_METHOD

END_FUNCTION_BLOCK

// TEST/TestPackage/Structure Samples/PRG02/TEMPLATES/Standard/Universal/Valve/FB_Bnet_Vlv_014
FUNCTION_BLOCK FB_Bnet_Vlv_014 EXTENDS FB_BACnet_View
VAR_INPUT
	bEnSfty			: BOOL;
	fValSfty		: REAL;
	bEnCrit			: BOOL;
	fValCrit		: REAL;
	fValPgm			: REAL;
END_VAR
VAR_OUTPUT
	fPresentValue	: REAL;
	bEvent			: BOOL;
END_VAR
VAR
	AO								: FB_BACnet_AO_IO5P := (
										iParent 				:= THIS^,
										sObjectName				:= '\/CMD01',
										sDescription			:= '\/Schaltbefehl',
										sDeviceType				:= 'Ventil',
										fResolution				:= 0.003051851,
										fScaleOffset			:= 0,
										eUnit					:= E_BA_Unit.eOther_Percent);
END_VAR

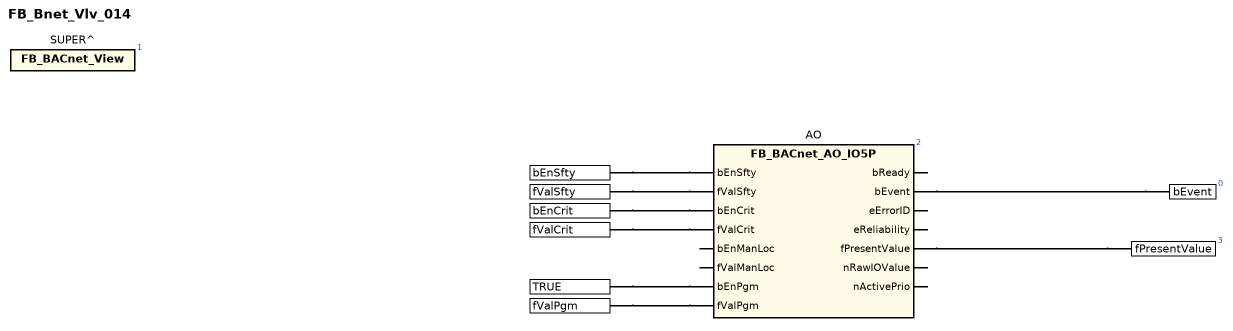
bEvent := AO.bEvent;
SUPER^(); // FB_BACnet_View
AO(
    bEnSfty := bEnSfty,
    fValSfty := fValSfty,
    bEnCrit := bEnCrit,
    fValCrit := fValCrit,
    bEnPgm := TRUE,
    fValPgm := fValPgm); // FB_BACnet_AO_IO5P
fPresentValue := AO.fPresentValue;

METHOD FB_init : BOOL
VAR_INPUT
	bInitRetains : BOOL; // if TRUE, the retain variables are initialized (warm start / cold start)
	bInCopyCode : BOOL;  // if TRUE, the instance afterwards gets moved into the copy code (online change)
END_VAR
sObjectName		:= '\/VLV01';
sDescription	:= '\/Ventil';
END_METHOD

END_FUNCTION_BLOCK

// TEST/TestPackage/Structure Samples/PRG02/MAIN_PRG02
PROGRAM MAIN_PRG02
VAR
	B01								: FB_BACnet_View		:= (							sObjectName := '\/B01',			sDescription :=	'Gebäude 1');
	B01_ISP01						: FB_BACnet_View		:= (iParent	:= B01,				sObjectName := '\/ISP01',		sDescription :=		'Informationsschwerpunkt 1');
	B01_ISP01_H						: FB_BACnet_View		:= (iParent	:= B01_ISP01,		sObjectName := '\/H',			sDescription :=			'Heizungsanlagen');
	B01_ISP01_H_HtgCir01			: FB_BA_HtgCir01		:= (iParent	:= B01_ISP01_H,		sObjectName := '\/HTG01',		sDescription :=				'Statischer Heizkreis 1');			// Hier ein Standard-Heizkreis
	B01_ISP01_H_HtgCir02			: FB_BA_HtgCir01		:= (iParent	:= B01_ISP01_H,		sObjectName := '\/HTG02',		sDescription :=				'Statischer Heizkreis 2');			// Hier ein Standard-Heizkreis
	B01_ISP01_H_HtgCir03			: FB_BA_HtgCir01		:= (iParent	:= B01_ISP01_H,		sObjectName := '\/HTG03',		sDescription :=				'Statischer Heizkreis 3');			// Hier ein Standard-Heizkreis
	B01_ISP01_H_HtgCirABC123		: FB_BA_HtgCirABC123	:= (iParent	:= B01_ISP01_H,		sObjectName := '\/HTG11',		sDescription :=				'Heizkreis Kantine');				// Hier ein angepasster Heizkreis
	B01_ISP01_H_HtgCirTZU555		: FB_BA_HtgCirTZU555	:= (iParent	:= B01_ISP01_H,		sObjectName := '\/HTG12',		sDescription :=				'Heizkreis Hausmeister',			// Hier ein angepasster Heizkreis + individualisierung
																Pu := (
																	Dst := (
																		ePolarity			:= E_BA_Polarity.eReverse),
																	BO := (
																		sActiveText			:= 'Bin an',
																		sInactiveText		:= 'Bin aus')
																));
	B01_ISP01_AC					: FB_BACnet_View		:= (iParent	:= B01_ISP01,		sObjectName := '\/AC',			sDescription			:= 'Lüftungsanlagen');
	B01_ISP01_AC_AC01				: FB_BA_AC01			:= (iParent	:= B01_ISP01_AC,	sObjectName := '\/APLT01',		sDescription				:= 'Lüftungsanlage 1');				// Hier eine Standard-Lüftung
	B01_ISP01_AC_AC02				: FB_BA_AC01			:= (iParent	:= B01_ISP01_AC,	sObjectName := '\/APLT02',		sDescription				:= 'Lüftungsanlage 2');				// Hier eine Standard-Lüftung
	B01_ISP01_AC_AC03				: FB_BA_AC01			:= (iParent	:= B01_ISP01_AC,	sObjectName := '\/APLT03',		sDescription				:= 'Lüftungsanlage 3');				// Hier eine Standard-Lüftung
	B01_ISP01_AC_AC04				: FB_BA_AC01			:= (iParent	:= B01_ISP01_AC,	sObjectName := '\/APLT04',		sDescription				:= 'Lüftungsanlage 4');				// Hier eine Standard-Lüftung
	B01_ISP01_AC_AC05				: FB_BA_AC01			:= (iParent	:= B01_ISP01_AC,	sObjectName := '\/APLT05',		sDescription				:= 'Lüftungsanlage 5');				// Hier eine Standard-Lüftung
END_VAR

B01();
B01_ISP01();
B01_ISP01_H();
B01_ISP01_H_HtgCir01();
B01_ISP01_H_HtgCir02();
B01_ISP01_H_HtgCir03();
B01_ISP01_H_HtgCirABC123();
B01_ISP01_H_HtgCirTZU555();
B01_ISP01_AC();
B01_ISP01_AC_AC01();
B01_ISP01_AC_AC02();
B01_ISP01_AC_AC03();
B01_ISP01_AC_AC04();
B01_ISP01_AC_AC05();

END_PROGRAM

// TEST/TestPackage/TEMPLATES/HeatSupply/HeatingCircuit/Plants/FB_Bnet_H_HtgCir_01
FUNCTION_BLOCK FB_Bnet_H_HtgCir_01 EXTENDS FB_BACnet_View
VAR_INPUT CONSTANT
	WthT							: FB_BACnet_AI_IO := (
										iParent 					:= THIS^,
										sObjectName					:= '\/WTHT',
										sDescription				:= '\/Aussentemperatur',
										sDeviceType					:= 'Temperatursensor',
										fResolution					:= 0.003051851,
										eUnit						:= E_BA_Unit.eTemperature_DegreesCelsius);
										
	FlWT							: FB_BACnet_AI_IO := (
										iParent 					:= THIS^,
										sObjectName					:= '\/TVL',
										sDescription				:= '\/Vorlauftemperatur',
										sDeviceType					:= 'Temperatursensor',
										fResolution					:= 0.003051851,
										eUnit						:= E_BA_Unit.eTemperature_DegreesCelsius);
	RtWT							: FB_BACnet_AI_IO := (
										iParent 					:= THIS^,
										sObjectName					:= '\/TRT',
										sDescription				:= '\/Rücklauftemperatur',
										sDeviceType					:= 'Temperatursensor',
										fResolution					:= 0.003051851,
										fScaleOffset				:= 0,
										eUnit						:= E_BA_Unit.eTemperature_DegreesCelsius);
										
	Sched							: FB_BACnet_SchedB := (
										iParent 					:= THIS^,
										sObjectName					:= '\/SCH01',
										sDescription				:= '\/Zeitschaltprogramm',
										tWeek						:= F_BACnet_SchedWeekly3xB(E_BA_Weekday.eMonday, E_BA_Weekday.eFriday, T#0H, FALSE, T#6H, TRUE, T#20H, FALSE));
										
	PID								: FB_BACnet_Loop := (
										iParent 					:= THIS^,
										sObjectName					:= '\/PID01',
										sDescription				:= '\/Vorlauftemperaturregler',
										eAction						:= E_BA_Action.eReverse,
										fPropertionalConstant		:= 1,
										fIntegralConstant			:= 180);	
										
	OpM								: FB_Bnet_H_OpM := (
										iParent 					:= THIS^);	
										
	SpG								: FB_Bnet_H_HtgCir_Sp := (
										iParent 					:= THIS^);	
										
	HtgLimit						: FB_Bnet_H_HtgCir_HtgLmt := (
										iParent 					:= THIS^);
										
	Vlv								: FB_Bnet_Vlv_013 := (
										iParent 					:= THIS^);	
										
	Pu								: FB_Bnet_Pu1st := (
										iParent 					:= THIS^);	
END_VAR
VAR // added by the converter: edge detectors and wires of the graphical bodies
    _w1 : ANY;
END_VAR

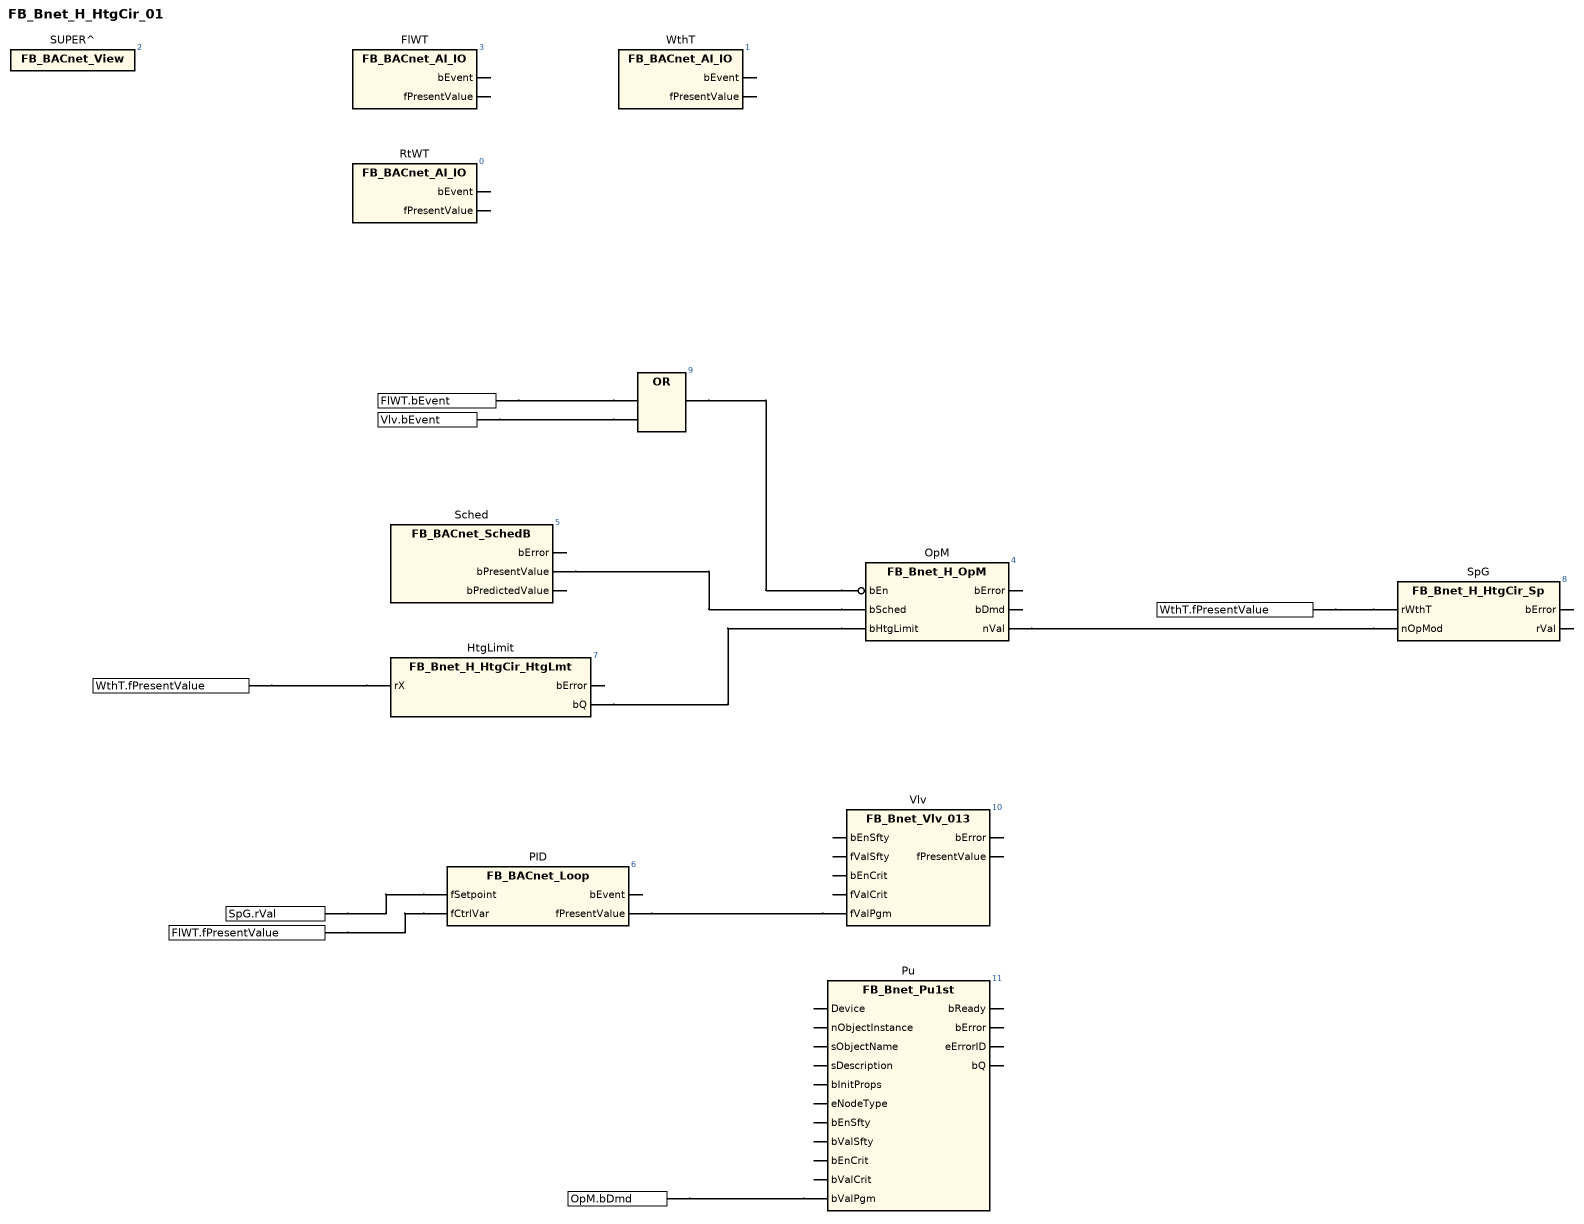
// note: 28 stored wires end on pins the file does not list and are not shown
RtWT(); // FB_BACnet_AI_IO
WthT(); // FB_BACnet_AI_IO
SUPER^(); // FB_BACnet_View
FlWT(); // FB_BACnet_AI_IO
OpM(bEn := NOT _w1, bSched := Sched.bPresentValue, bHtgLimit := HtgLimit.bQ); // FB_Bnet_H_OpM
Sched(); // FB_BACnet_SchedB
PID(fSetpoint := SpG.rVal, fCtrlVar := FlWT.fPresentValue); // FB_BACnet_Loop
HtgLimit(rX := WthT.fPresentValue); // FB_Bnet_H_HtgCir_HtgLmt
SpG(rWthT := WthT.fPresentValue, nOpMod := OpM.nVal); // FB_Bnet_H_HtgCir_Sp
_w1 := FlWT.bEvent OR Vlv.bEvent;
Vlv(fValPgm := PID.fPresentValue); // FB_Bnet_Vlv_013
Pu(bValPgm := OpM.bDmd); // FB_Bnet_Pu1st

METHOD FB_init : BOOL
VAR_INPUT
	bInitRetains : BOOL; // if TRUE, the retain variables are initialized (warm start / cold start)
	bInCopyCode : BOOL;  // if TRUE, the instance afterwards gets moved into the copy code (online change)
END_VAR
sObjectName		:= '\/HCR01';
sDescription	:= '\/Heizkreis';

Pu.BO.sObjectName := '\/XXXtest';
END_METHOD

END_FUNCTION_BLOCK

// TEST/TestPackage/TEMPLATES/Internal/FB_BA_Server_NC01
// Notification Classes (Sample 01: Beckhoff)	
FUNCTION_BLOCK FB_BA_Server_NC01 EXTENDS FB_BACnet_View
VAR CONSTANT
	iAlarmModeFirst		: INT		:= 1;
	iAlarmModeLast		: INT		:= 3;
END_VAR
VAR
	// Event Typ "Alarm":
	fbNCAlm_LifeSafety		: ARRAY[iAlarmModeFirst .. iAlarmModeLast] OF FB_BACnet_NC := [
								(
									iParent									:= THIS^,
									nObjectInstance							:= 12,
									nNotificationClass						:= 12,
									sObjectName								:= '\/NC12',
									sDescription							:= '\/Meldeklasse - Alarm Lebensgefahr (Einfach)',
									bAckRequired							:= [ TRUE, TRUE, FALSE ],
									nPriority								:= [ 10, 11, 12 ]),
								(
									iParent									:= THIS^,
									nObjectInstance							:= 11,
									nNotificationClass						:= 11,
									sObjectName								:= '\/NC11',
									sDescription							:= '\/Meldeklasse - Alarm Lebensgefahr (Standard)',
									bAckRequired							:= [ TRUE, TRUE, FALSE ],
									nPriority								:= [ 13, 14, 15 ]),
								(
									iParent									:= THIS^,
									nObjectInstance							:= 10,
									nNotificationClass						:= 10,
									sObjectName								:= '\/NC10',
									sDescription							:= '\/Meldeklasse - Alarm Lebensgefahr (Erweitert)',
									bAckRequired							:= [ TRUE, TRUE, TRUE ],
									nPriority								:= [ 16, 17, 18 ])
							];
							
	fbNCAlm_Technical		: ARRAY[iAlarmModeFirst .. iAlarmModeLast] OF FB_BACnet_NC := [
								(
									iParent									:= THIS^,
									nObjectInstance							:= 22,
									nNotificationClass						:= 22,
									sObjectName								:= '\/NC22',
									sDescription							:= '\/Meldeklasse - Technischer Alarm (Einfach)',
									bAckRequired							:= [ TRUE, TRUE, FALSE ],
									nPriority								:= [ 20, 21, 22 ]),
								(
									iParent									:= THIS^,
									nObjectInstance							:= 21,
									nNotificationClass						:= 21,
									sObjectName								:= '\/NC21',
									sDescription							:= '\/Meldeklasse - Technischer Alarm (Standard)',
									bAckRequired							:= [ TRUE, TRUE, FALSE ],
									nPriority								:= [ 23, 24, 25 ]),
								(
									iParent									:= THIS^,
									nObjectInstance							:= 20,
									nNotificationClass						:= 20,
									sObjectName								:= '\/NC20',
									sDescription							:= '\/Meldeklasse - Technischer Alarm (Erweitert)',
									bAckRequired							:= [ TRUE, TRUE, TRUE ],
									nPriority								:= [ 26, 27, 28 ])
							];
							
	// Event Typ "Disturb":
	fbNCDstb				: ARRAY[iAlarmModeFirst .. iAlarmModeLast] OF FB_BACnet_NC := [
								(
									iParent									:= THIS^,
									nObjectInstance							:= 52,
									nNotificationClass						:= 52,
									sObjectName								:= '\/NC52',
									sDescription							:= '\/Meldeklasse - Störung (Einfach)',
									bAckRequired							:= [ TRUE, TRUE, FALSE ],
									nPriority								:= [ 50, 51, 52 ]),
								(
									iParent									:= THIS^,
									nObjectInstance							:= 51,
									nNotificationClass						:= 51,
									sObjectName								:= '\/NC51',
									sDescription							:= '\/Meldeklasse - Störung (Standard)',
									bAckRequired							:= [ TRUE, TRUE, FALSE ],
									nPriority								:= [ 53, 54, 55 ]),
								(
									iParent									:= THIS^,
									nObjectInstance							:= 50,
									nNotificationClass						:= 50,
									sObjectName								:= '\/NC50',
									sDescription							:= '\/Meldeklasse - Störung (Erweitert)',
									bAckRequired							:= [ TRUE, TRUE, TRUE ],
									nPriority								:= [ 56, 57, 58 ])
							];
							
	// Event Typ "Maintenance":
	fbNCMntn				: ARRAY[iAlarmModeFirst .. iAlarmModeLast] OF FB_BACnet_NC := [
								(
									iParent									:= THIS^,
									nObjectInstance							:= 92,
									nNotificationClass						:= 92,
									sObjectName								:= '\/NC92',
									sDescription							:= '\/Meldeklasse - Wartung (Einfach)',
									bAckRequired							:= [ TRUE, TRUE, FALSE ],
									nPriority								:= [ 90, 91, 92 ]),
								(
									iParent									:= THIS^,
									nObjectInstance							:= 91,
									nNotificationClass						:= 91,
									sObjectName								:= '\/NC91',
									sDescription							:= '\/Meldeklasse - Wartung (Standard)',
									bAckRequired							:= [ TRUE, TRUE, FALSE ],
									nPriority								:= [ 93, 94, 95 ]),
								(
									iParent									:= THIS^,
									nObjectInstance							:= 90,
									nNotificationClass						:= 90,
									sObjectName								:= '\/NC90',
									sDescription							:= '\/Meldeklasse - Wartung (Erweitert)',
									bAckRequired							:= [ TRUE, TRUE, TRUE ],
									nPriority								:= [ 96, 97, 98 ])
							];
							
	// Event Typ "Notification":
	fbNCNtfy				: ARRAY[iAlarmModeFirst .. iAlarmModeLast] OF FB_BACnet_NC := [
								(
									iParent									:= THIS^,
									nObjectInstance							:= 132,
									nNotificationClass						:= 132,
									sObjectName								:= '\/NC132',
									sDescription							:= '\/Meldeklasse - Benachrichtigung (Einfach)',
									bAckRequired							:= [ TRUE, TRUE, FALSE ],
									nPriority								:= [ 130, 131, 132 ]),
								(
									iParent									:= THIS^,
									nObjectInstance							:= 131,
									nNotificationClass						:= 131,
									sObjectName								:= '\/NC131',
									sDescription							:= '\/Meldeklasse - Benachrichtigung (Standard)',
									bAckRequired							:= [ TRUE, TRUE, FALSE ],
									nPriority								:= [ 133, 134, 135 ]),
								(
									iParent									:= THIS^,
									nObjectInstance							:= 130,
									nNotificationClass						:= 130,
									sObjectName								:= '\/NC130',
									sDescription							:= '\/Meldeklasse - Benachrichtigung (Erweitert)',
									bAckRequired							:= [ TRUE, TRUE, TRUE ],
									nPriority								:= [ 136, 137, 138 ])
							];
							
	// Event Typ "Other":	
	fbNCOthr				: ARRAY[iAlarmModeFirst .. iAlarmModeLast] OF FB_BACnet_NC := [
								(
									iParent									:= THIS^,
									nObjectInstance							:= 182,
									nNotificationClass						:= 182,
									sObjectName								:= '\/NC182',
									sDescription							:= '\/Meldeklasse - Sonstiges (Einfach)',
									bAckRequired							:= [ TRUE, TRUE, FALSE ],
									nPriority								:= [ 180, 181, 182 ]),
								(
									iParent									:= THIS^,
									nObjectInstance							:= 181,
									nNotificationClass						:= 181,
									sObjectName								:= '\/NC181',
									sDescription							:= '\/Meldeklasse - Sonstiges (Standard)',
									bAckRequired							:= [ TRUE, TRUE, FALSE ],
									nPriority								:= [ 183, 184, 185 ]),
								(
									iParent									:= THIS^,
									nObjectInstance							:= 180,
									nNotificationClass						:= 180,
									sObjectName								:= '\/NC180',
									sDescription							:= '\/Meldeklasse - Sonstiges (Erweitert)',
									bAckRequired							:= [ TRUE, TRUE, TRUE ],
									nPriority								:= [ 186, 187, 188 ])
							];
END_VAR
VAR
	iValTmp						: INT;
	iTemp						: INT;
END_VAR

SUPER^();

FOR iTemp := iAlarmModeFirst TO iAlarmModeLast DO
	fbNCAlm_LifeSafety[iTemp]();
	fbNCAlm_Technical[iTemp]();
	fbNCDstb[iTemp]();
	fbNCMntn[iTemp]();
	fbNCNtfy[iTemp]();
	fbNCOthr[iTemp]();
END_FOR

END_FUNCTION_BLOCK

// TEST/TestPackage/TestFBs/RT/FB_ArrayHtgCir
FUNCTION_BLOCK FB_ArrayHtgCir EXTENDS FB_BACnet_View
VAR_INPUT
	iCycleCount				: UINT;
END_VAR
VAR
	iTemp					: INT;
	fbPlants				: ARRAY [1..MAX_PLANT] OF FB_Bnet_H_HtgCir_01;

	iCycleMOD				: UINT := 1;
	iLoopTo					: INT := MAX_PLANT;
END_VAR
VAR CONSTANT
	//MAX_PLANT				: INT := 29;			// Entspricht 1021 Ibjekte
	MAX_PLANT				: INT := 1;
END_VAR

SUPER^();

IF ((iCycleCount MOD iCycleMOD) = 0) THEN
	FOR iTemp := 1 TO iLoopTo DO
		fbPlants[iTemp]();
	END_FOR
END_IF

METHOD FB_init : BOOL
VAR_INPUT
	bInitRetains : BOOL; // if TRUE, the retain variables are initialized (warm start / cold start)
	bInCopyCode : BOOL;  // if TRUE, the instance afterwards gets moved into the copy code (online change)
END_VAR
sObjectName		:= 'Test Heizkreise';
sDescription	:= 'Array mit vielen Heizkreisen';

FOR iTemp := 1 TO MAX_PLANT DO
	fbPlants[iTemp].Parent			:= THIS^;
	fbPlants[iTemp].sObjectName 	:= CONCAT('HtgCir', TO_STRING(iTemp));
	fbPlants[iTemp].sDescription	:= CONCAT('Heizkreis ', TO_STRING(iTemp));
END_FOR
END_METHOD

END_FUNCTION_BLOCK

// TEST/TestPackage/TestFBs/RT/FB_ArrayTest
FUNCTION_BLOCK FB_ArrayTest EXTENDS FB_BACnet_View
VAR_INPUT
	iCycleCount				: UINT;
END_VAR
VAR					
	iTemp					: INT;
	BVObjects				: ARRAY [1..MAX_OBJECT] OF FB_BACnet_BV;

	iCycleMOD				: UINT := 1;
	iLoopTo					: INT := MAX_OBJECT;
END_VAR
VAR CONSTANT
	MAX_OBJECT : INT := 1000;
END_VAR

SUPER^();

IF ((iCycleCount MOD iCycleMOD) = 0) THEN
	FOR iTemp := 1 TO iLoopTo DO
		BVObjects[iTemp]();
	END_FOR
END_IF

METHOD FB_init : BOOL
VAR_INPUT
	bInitRetains : BOOL; // if TRUE, the retain variables are initialized (warm start / cold start)
	bInCopyCode : BOOL;  // if TRUE, the instance afterwards gets moved into the copy code (online change)
END_VAR
sObjectName		:= 'TestArray';
sDescription	:= 'Array mit vielen Objekten';

FOR iTemp := 1 TO MAX_OBJECT DO
	BVObjects[iTemp].Parent						:= THIS^;
	BVObjects[iTemp].sObjectName 				:= CONCAT('BV üäß', TO_STRING(iTemp));
	BVObjects[iTemp].sDescription				:= CONCAT('Binary Value üäß ', TO_STRING(iTemp));
	
	BVObjects[iTemp].sActiveText				:= '€ ÄÄÄ üß';
	BVObjects[iTemp].sInactiveText				:= 'Money money $$ ÄÄÄ üß';
END_FOR
END_METHOD

END_FUNCTION_BLOCK

// TEST/TestPackage/TestFBs/FB_ClientTest
FUNCTION_BLOCK FB_ClientTest
VAR_INPUT CONSTANT
	AV_1 : FB_BACnetRM_AV := (Client:=Client,nObjectInstance:=1);
	AV_2 : FB_BACnetRM_AV := (Client:=Client,nObjectInstance:=2);
	AV_3 : FB_BACnetRM_AV := (Client:=Client,nObjectInstance:=3);
	AV_4 : FB_BACnetRM_AV := (Client:=Client,nObjectInstance:=4);
	AV_5 : FB_BACnetRM_AV := (Client:=Client,nObjectInstance:=5);
	AV_6 : FB_BACnetRM_AV := (Client:=Client,nObjectInstance:=6);
	AV_7 : FB_BACnetRM_AV := (Client:=Client,nObjectInstance:=7);
	AV_8 : FB_BACnetRM_AV := (Client:=Client,nObjectInstance:=8);
	AV_9 : FB_BACnetRM_AV := (Client:=Client,nObjectInstance:=9);
	AV_10: FB_BACnetRM_AV := (Client:=Client,nObjectInstance:=10);
	AV_11: FB_BACnetRM_AV := (Client:=Client,nObjectInstance:=11);
	AV_12: FB_BACnetRM_AV := (Client:=Client,nObjectInstance:=12);
END_VAR
VAR
	Client : FB_BACnet_Client := (eReadMode:=E_BACnet_CommMode.eRp);
END_VAR

Client();
AV_1();
AV_2();
AV_3();
AV_4();
AV_5();
AV_6();
AV_7();
AV_8();
AV_9();
AV_10();
AV_11();
AV_12();

END_FUNCTION_BLOCK

// TEST/TestPackage/_MAIN
PROGRAM _MAIN
VAR
	wDummy			AT %I*	: WORD;
	
	bKillMe11				: BOOL;
	bKillMe12				: BOOL;
END_VAR
VAR
	bInit					: BOOL := TRUE;
	nCycles					: UDINT;
END_VAR
VAR
	bManualWritePersistent	: BOOL;
	tAutoWritePersistent	: TON						:= (PT := T#20S);
	wPersistentData			: FB_WritePersistentData	:= (PORT:=TwinCAT_SystemInfoVarList._AppInfo.AdsPort, TMOUT:=T#1S, MODE:=E_PersistentMode.SPDM_2PASS);
END_VAR

nCycles := (nCycles+1);
IF (bInit) THEN
	bInit := FALSE;
END_IF

// Persistent data:
tAutoWritePersistent(IN := (NOT tAutoWritePersistent.Q));
IF (bManualWritePersistent) OR (tAutoWritePersistent.Q) THEN
	bManualWritePersistent := FALSE;
	wPersistentData(START:=TRUE);
ELSE
	wPersistentData();
	IF (NOT wPersistentData.BUSY) THEN
		wPersistentData.START:=FALSE;
	END_IF
END_IF

// Sample programs:
// Uncomment to execute samples:
//////////////////////////////////////////////////

//CLIENT();
//PLANT_DEMO();
//MAIN_PRG02();
//PERFORMANCE();
//PERFORMANCE_MIX();
//RT();

END_PROGRAM

// TEST/TestPackage/PLANT_DEMO
PROGRAM PLANT_DEMO
VAR
	fbStatHeatingCir	: FB_Bnet_H_HtgCir_01		:= (sObjectName				:= 'HTGCIR01',
														sDescription			:= '\/Statische Heizung',
														Pu := (
															sObjectName			:= '\/TEST01_PU01',
															Dst := (
																sObjectName		:= '\/DST01')));
																
	fbFlHeatingCir		: FB_Bnet_H_HtgCir_01		:= (sObjectName				:= 'HTGCIR02',
														sDescription			:= '\/Fußbodenheizung');
																
	fbRoom3				: FB_Bnet_H_HtgCir_01		:= (sObjectName				:= 'HTGCIR03',
														sDescription			:= '\/Heizung Raum 3');
END_VAR

fbStatHeatingCir();
fbFlHeatingCir();
fbRoom3();

METHOD FB_init : BOOL
VAR_INPUT
	bInitRetains : BOOL; // if TRUE, the retain variables are initialized (warm start / cold start)
	bInCopyCode : BOOL;  // if TRUE, the instance afterwards gets moved into the copy code (online change)
END_VAR
fbStatHeatingCir.Pu.sObjectName			:= '\/TEST01_PU01';
fbStatHeatingCir.Pu.sObjectName			:= '\/TEST01_PU01';
fbStatHeatingCir.Pu.sObjectName			:= '\/TEST01_PU01';
fbStatHeatingCir.Pu.sObjectName			:= '\/TEST01_PU01';
fbStatHeatingCir.Pu.sObjectName			:= '\/TEST01_PU01';
END_METHOD

END_PROGRAM

// TEST/TestPackage/PERFORMANCE
PROGRAM PERFORMANCE
// Test für RT-Objekte:
VAR
	//fbHtgCirArray : FB_ArrayHtgCir;
	fbObjArray : FB_ArrayTest;
	
	bStop : BOOL;
END_VAR


// Test für RT-Objekte:
//fbHtgCirArray();
IF NOT bStop THEN
	fbObjArray();
END_IF

END_PROGRAM

// TEST/TestPackage/RT
// Dieses Programm testet die RT-Bausteine, welche der LIB-Variante nachempfunden sind.
PROGRAM RT
VAR
	bKillMe1 : BOOL;
	bKillMe2 : BOOL;
	_hRes : HRESULT;
	tTemp : T_MaxString;
END_VAR
VAR_INPUT
	nLibNode_UpdateCount				: UDINT;
	fbLibNode							: FB_BACnet_View := (
											eNodeType								:= E_BACnet_NodeType.eArea,
											sObjectName								:= '\/LibNde',
											sDescription							:= '\/Test RT-Lib Node');
END_VAR
// --- Analog: ---------------------------------------------------------------------------------------------------------------------------------------
VAR_INPUT
	fbANode								: FB_BACnet_View := (
											iParent									:= fbLibNode,
											eNodeType								:= E_BACnet_NodeType.eArea,
											sObjectName								:= '\/A',
											sDescription							:= '\/Analog');
											
	AV									: FB_BACnet_AV := (
											iParent									:= fbANode,
											nObjectInstance							:= 111,
											sObjectName								:= '\/AV01',
											sDescription							:= '\/Analog Value Test 1 öäü',
											eUnit									:= E_BA_Unit.eOther_Percent,
											bHighLimitEnable						:= TRUE,
											fHighLimitValue							:= 50,
											bLowLimitEnable							:= TRUE,
											fLowLimitValue							:= 10,
											nNotificationClass						:= 11,
											bEventEnable							:= [ TRUE, TRUE, FALSE ],
											sEventMessageTextsConfig				:= [ '\/Ausgelöst', '\/Fehler', '\/Normal' ]);

	// Intention:						Value
	// Priorities						5P
	AV5P_TestEnSfty				AT %I*	: BOOL; // Test: Safety ist von PLC aus immer beschaltet
	AV5P								: FB_BACnet_AV_5P := (
											iParent									:= fbANode,
											sDescription							:= '\/Analog Value 5Prio',
											eUnit									:= E_BA_Unit.eOther_Percent);
											
	// Intention:						Value for Display
	// Operation:						Display
	AVDsp								: FB_BACnet_AV_Disp := (
											iParent									:= fbANode,
											sDescription							:= '\/Test AV Display',
											eUnit									:= E_BA_Unit.eOther_Percent);	
	
	// Intention:						Value for Setpoint
	// Operation:						Setpoint
	AVSp								: FB_BACnet_AV_Setp := (
											iParent									:= fbANode,
											sDescription							:= '\/Test AV Setpoint',
											eUnit									:= E_BA_Unit.eTime_Hours,
											fValue									:= 168);

	AI_TSenRaw_State			AT %I*	: USINT;
	AI_TSenRaw_DataIn			AT %I*	: INT;
	AI_TSenRaw							: FB_BACnet_AI_Raw := (
											iParent									:= fbANode,
											sDescription							:= '\/Test AI Fühler (Raw)',
											sDeviceType								:= 'Fühler',
											eUnit									:= E_BA_Unit.eOther_Percent,
											fResolution								:= 0.003814755,
											fScaleOffset							:= 0.0,
											fHighLimitValue							:= 150,
											fLowLimitValue							:= -500,
											nNotificationClass						:= 10,
											bEventEnable							:= [ TRUE, TRUE, FALSE ],
											sEventMessageTextsConfig				:= [ '\/Ausgelöst', '\/Fehler', '\/Normal' ]);

	// Intention:						Input
	// Hardware:						Process
	AI_TSenProc_Value					: REAL := 50.0;
	AI_TSenProc							: FB_BACnet_AI := (
											iParent									:= fbANode,
											sDescription							:= '\/Test AI (Prozesswert)',
											eUnit									:= E_BA_Unit.eOther_Percent,
											fHighLimitValue							:= 150,
											fLowLimitValue							:= -500,
											nNotificationClass						:= 10,
											bEventEnable							:= [ TRUE, TRUE, FALSE ],
											sEventMessageTextsConfig				:= [ '\/Ausgelöst', '\/Fehler', '\/Normal' ]);

	// Intention:						Input
	// Hardware:						I/O
	AI_TSenIO							: FB_BACnet_AI_IO := (
											iParent									:= fbANode,
											sDescription							:= '\/Test AI Fühler (IO)',
											sDeviceType								:= 'Fühler',
											eUnit									:= E_BA_Unit.eOther_Percent,
											fResolution								:= 0.003814755,
											fScaleOffset							:= 0.0,
											fHighLimitValue							:= 150,
											fLowLimitValue							:= -500,
											nNotificationClass						:= 10,
											bEventEnable							:= [ TRUE, TRUE, FALSE ],
											sEventMessageTextsConfig				:= [ '\/Ausgelöst', '\/Fehler', '\/Normal' ]);

	// Intention:						Input for Display
	// Operation:						Display
	// Hardware:						I/O
	// Parameter:						EventDetectionEnable = FALSE
	AIDsp_TSenIO						: FB_BACnet_AI_IO := (
											iParent									:= fbANode,
											sDescription							:= '\/Test AI Display Fühler (IO)',
											sDeviceType								:= 'Fühler',
											eUnit									:= E_BA_Unit.eOther_Percent,
											bEventDetectionEnable					:= FALSE);

	AO_CmdRaw_Out				AT %Q*	: INT;
	AO_CmdRaw							: FB_BACnet_AO_Raw := (
											iParent									:= fbANode,
											sDescription							:= '\/Befehl AO (Raw)',
											sDeviceType								:= 'Ausgang',
											eUnit									:= E_BA_Unit.eOther_Percent,
											fResolution								:= 0.003051851,
											fScaleOffset							:= 0.0,
											fHighLimitValue							:= 150,
											fLowLimitValue							:= -50,
											nNotificationClass						:= 10,
											bEventEnable							:= [ TRUE, TRUE, FALSE ],
											sEventMessageTextsConfig				:= [ '\/Ausgelöst', '\/Fehler', '\/Normal' ]);

	AO_CmdIORaw							: FB_BACnet_AO_Raw := (
											iParent									:= fbANode,
											sDescription							:= '\/Befehl AO (IO)',
											sDeviceType								:= 'Ausgang',
											eUnit									:= E_BA_Unit.eOther_Percent,
											fResolution								:= 0.003051851,
											fScaleOffset							:= 0.0,
											fHighLimitValue							:= 150,
											fLowLimitValue							:= -50,
											nNotificationClass						:= 10,
											bEventEnable							:= [ TRUE, TRUE, FALSE ],
											sEventMessageTextsConfig				:= [ '\/Ausgelöst', '\/Fehler', '\/Normal' ]);

	AO_CmdRaw5P_State			AT %I*	: USINT;
	AO_CmdRaw5P_Out				AT %Q*	: INT;
	AO_CmdRaw5P							: FB_BACnet_AO_Raw5P := (
											iParent									:= fbANode,
											sDescription							:= '\/Analog Befehl 5Prio (Raw)',
											eUnit									:= E_BA_Unit.eOther_Percent);

	// Intention:						Output
	// Hardware:						I/O
	// Priorities						5P
	AO_CmdIO5P							: FB_BACnet_AO_IO5P := (
											iParent									:= fbANode,
											sDescription							:= '\/Analog Befehl 5Prio (IO)',
											eUnit									:= E_BA_Unit.eOther_Percent);

	// Intention:						Output for Display
	// Operation:						Display
	// Hardware:						I/O
	// Parameter:						EventDetectionEnable = FALSE
	AODisp_CmdIO5P						: FB_BACnet_AO_IO5P := (
											iParent									:= fbANode,
											sDescription							:= '\/Analog Befehl 5Prio Display (IO)',
											eUnit									:= E_BA_Unit.eOther_Percent,
											bEventDetectionEnable					:= FALSE);
											
	AO_CmdIO							: FB_BACnet_AO_IO := (
											iParent									:= fbANode,
											sDescription							:= '\/Analog Befehl (IO)',
											eUnit									:= E_BA_Unit.eOther_Percent);
END_VAR
// --- Binary: ---------------------------------------------------------------------------------------------------------------------------------------
VAR_INPUT
	fbBNode								: FB_BACnet_View := (
											iParent									:= fbLibNode,
											eNodeType								:= E_BACnet_NodeType.eArea,
											sObjectName								:= '\/B',
											sDescription							:= '\/Binary');
											
	BV									: FB_BACnet_BV := (
											iParent									:= fbBNode,
											nObjectInstance							:= 99,
											sDescription							:= '\/Test BV',
											bAlarmValue								:= FALSE);

	// Intention:						Value
	// Priorities						5P
	BV5P								: FB_BACnet_BV_5P := (
											iParent									:= fbBNode,
											sDescription							:= '\/Binary Value 5Prio');
											
	// Intention:						Value for Display
	// Operation:						Display
	BVDsp								: FB_BACnet_BV_Disp := (
											iParent									:= fbBNode,
											sDescription							:= '\/Test BV Display',
											sInactiveText							:= 'Aus',
											sActiveText								:= 'Ein');
	
	// Intention:						Value for Setpoint
	// Operation:						Setpoint
	BVSp								: FB_BACnet_BV_Setp := (
											iParent									:= fbBNode,
											sDescription							:= '\/Test BV Setpoint',
											sInactiveText							:= 'Aus',
											sActiveText								:= 'Ein',
											bValue									:= TRUE);

	BI_DstbRaw_In				AT %I*	: BOOL;
	BI_DstbRaw							: FB_BACnet_BI_Raw := (
											iParent									:= fbBNode,
											sDescription							:= '\/Test BI Disturb (Raw)',
											sDeviceType								:= 'Sicherung',
											sInactiveText							:= 'Normal',
											sActiveText								:= 'Ausgelöst',
											ePolarity								:= E_BA_Polarity.eReverse,
											nNotificationClass						:= 10,
											bEventEnable							:= [ TRUE, TRUE, FALSE ],
											sEventMessageTextsConfig				:= [ '\/Ausgelöst', '\/Fehler', '\/Normal' ]);
											
	// Intention:						Input
	// Hardware:						I/O
	BI_DstbIO							: FB_BACnet_BI_IO := (
											iParent									:= fbBNode,
											sDescription							:= '\/Test BI Disturb (IO)',
											sDeviceType								:= 'Sicherung',
											sInactiveText							:= 'Normal',
											sActiveText								:= 'Ausgelöst',
											ePolarity								:= E_BA_Polarity.eReverse,
											nNotificationClass						:= 10,
											bEventEnable							:= [ TRUE, TRUE, FALSE ],
											sEventMessageTextsConfig				:= [ '\/Ausgelöst', '\/Fehler', '\/Normal' ]);

	// Intention:						Input for Display
	// Operation:						Display
	// Hardware:						I/O
	// Parameter:						EventDetectionEnable = FALSE
	BIDsp_SwiIO							: FB_BACnet_BI_IO := (
											iParent									:= fbBNode,
											sDescription							:= '\/Test BI Schalter Display (IO)',
											sDeviceType								:= 'Sicherung',
											sInactiveText							:= 'Normal',
											sActiveText								:= 'Ausgelöst',
											ePolarity								:= E_BA_Polarity.eReverse,
											bEventDetectionEnable					:= FALSE);

	BO_CmdRaw_Out				AT %Q*	: BOOL;
	BO_CmdRaw							: FB_BACnet_BO_Raw := (
											iParent									:= fbBNode,
											sDescription							:= '\/Test BO Befehl (Raw)',
											sInactiveText							:= 'Aus',
											sActiveText								:= 'Ein');
											
	BO_CmdIO							: FB_BACnet_BO_IO := (
											iParent									:= fbBNode,
											sDescription							:= '\/Test BO Befehl (IO)',
											sInactiveText							:= 'Aus',
											sActiveText								:= 'Ein');

	BO_CmdRaw5P_Feedback		AT %I*	: BOOL;
	BO_CmdRaw5P_OverrIO			AT %I*	: BOOL;
	BO_CmdRaw5P_Out				AT %Q*	: BOOL;
	BO_CmdRaw5P							: FB_BACnet_BO_Raw5P := (
											iParent									:= fbBNode,
											sDescription							:= '\/Test BO Befehl 5Prio (Raw)',
											sInactiveText							:= 'Aus',
											sActiveText								:= 'Ein',
											nTimeDelay								:= 3);
											
	// Intention:						Output
	// Hardware:						I/O
	// Priorities						5P
	BO_CmdIO5P							: FB_BACnet_BO_IO5P := (
											iParent									:= fbBNode,
											sDescription							:= '\/Test BO Befehl 5Prio (IO)',
											sInactiveText							:= 'Aus',
											sActiveText								:= 'Ein',
											nTimeDelay								:= 3);
											
	// Intention:						Output for Display
	// Operation:						Display
	// Hardware:						I/O
	// Parameter:						EventDetectionEnable = FALSE
	BODisp_CmdIO5P						: FB_BACnet_BO_IO5P := (
											iParent									:= fbBNode,
											sDescription							:= '\/Test BO Befehl 5Prio Display (IO)',
											sInactiveText							:= 'Aus',
											sActiveText								:= 'Ein',
											bEventDetectionEnable					:= FALSE);
END_VAR
// --- Multistate: ---------------------------------------------------------------------------------------------------------------------------------------
VAR_INPUT
	fbMNode								: FB_BACnet_View := (
											iParent									:= fbLibNode,
											eNodeType								:= E_BACnet_NodeType.eArea,
											sObjectName								:= '\/M',
											sDescription							:= '\/Multistate');
											
	MV									: FB_BACnet_MV := (
											iParent									:= fbMNode,
											nObjectInstance							:= 99,
											sDescription							:= '\/Test MV',
											nAlarmValues							:= [ 1, 2 ],
											nFaultValues							:= [ 3 ],
										//	sStateText								:= [ 'Aus', 'Stufe 1', 'Stufe 2']);
										//	sStateText								:= [ 'Aus', 'Stufe 1', 'Stufe 2', 'Stufe 3', 'Stufe 4', 'Stufe 5', 'Stufe 6', 'Stufe 7', 'Stufe 8', 'Stufe 9', 'Stufe 10', 'Stufe 11', 'Stufe 12', 'Stufe 13', 'Stufe 14', 'Stufe 15' ]);
											sStateText								:= [ 'Aus', 'Stufe 1', 'Stufe 2', 'Stufe 3', 'Stufe 4', 'Stufe 5', 'Stufe 6', 'Stufe 7', 'Stufe 8', 'Stufe 9', 'Stufe 10' ]);

	// Intention:						Value
	// Priorities						5P
	MV5P								: FB_BACnet_MV_5P := (
											iParent									:= fbMNode,
											sDescription							:= '\/Test MV 5Prio',
											sStateText								:= [ 'Aus', 'Stufe 1', 'Stufe 2' ]);

	// Intention:						Value for Display
	// Operation:						Display
	MVDsp								: FB_BACnet_MV_Disp := (
											iParent									:= fbMNode,
											sDescription							:= '\/Test MV Display',
											sStateText								:= [ 'Wert 11', 'Wert 22' ]);
	
	// Intention:						Value for Setpoint
	// Operation:						Setpoint
	MVSp								: FB_BACnet_MV_Setp := (
											iParent									:= fbMNode,
											sDescription							:= '\/Test MV Display',
											sStateText								:= [ 'Auto', 'Aus', 'Ein' ],
											nValue									:= 2);

	MI_StateRaw_In						: UDINT;
	MI_StateRaw							: FB_BACnet_MI_Raw := (
											iParent									:= fbMNode,
											sDescription							:= '\/Test MI State (Raw)',
											sDeviceType								:= 'Gerät',
											sStateText								:= [ 'Störung 1', 'Störung 2', 'Fehler', 'Normal' ],
											nAlarmValues							:= [ 1, 2 ],
											nFaultValues							:= [ 3 ],
											nNotificationClass						:= 10,
											bEventEnable							:= [ TRUE, TRUE, FALSE ],
											sEventMessageTextsConfig				:= [ '\/Ausgelöst', '\/Fehler', '\/Normal' ]);

	// Intention:						Input
	// Hardware:						I/O
	MI_StateIO							: FB_BACnet_MI_IO := (
											iParent									:= fbMNode,
											sDescription							:= '\/Test MI State (IO)',
											sDeviceType								:= 'Gerät',
											sStateText								:= [ 'Aus', 'Stufe 1', 'Stufe 2', 'Stufe 3', 'Stufe 4' ],
											nAlarmValues							:= [ 3, 4 ],
											nFaultValues							:= [ 5 ],
											nNotificationClass						:= 10,
											sEventMessageTextsConfig				:= [ '\/Ausgelöst', '\/Fehler', '\/Normal' ]
										);
										
	// Intention:						Input for Display
	// Operation:						Display
	// Hardware:						I/O
	// Parameter:						EventDetectionEnable = FALSE
	MIDsp_Swi_StateRaw_In				: UDINT;
	MIDsp_Swi_StateRaw					: FB_BACnet_MI_Raw := (
											iParent									:= fbMNode,
											sDescription							:= '\/Test MI State (Raw)',
											sDeviceType								:= 'Gerät',
											sStateText								:= [ 'Störung 1', 'Störung 2', 'Fehler', 'Normal' ],
											bEventDetectionEnable					:= FALSE);

	MO_CmdRaw_Out						: UDINT;
	MO_CmdRaw							: FB_BACnet_MO_Raw := (
											iParent									:= fbMNode,
											sDescription							:= '\/Test MO Befehl (Raw)',
											sStateText								:= [ 'Stufe 1', 'Stufe 2', 'Aus' ]);

	// Intention:						Output
	// Hardware:						I/O
	// Priorities						5P
	MO_Raw5P_Out						: UDINT;
	MO_Raw5P							: FB_BACnet_MO_Raw5P := (
											iParent									:= fbMNode,
											sDescription							:= '\/Test MO Befehl 5Prio (Raw)',
											sStateText								:= [ 'Stufe 1', 'Stufe 2', 'Aus' ]);

	MODisp_Raw5P_Out					: UDINT;
	MODisp_Raw5P						: FB_BACnet_MO_Raw5P := (
											iParent									:= fbMNode,
											sDescription							:= '\/Test MO Befehl 5Prio (Raw)',
											sStateText								:= [ 'Stufe 1', 'Stufe 2', 'Aus' ],
											bEventDetectionEnable					:= FALSE);
											

	// Intention:						Output for Display
	// Operation:						Display
	// Hardware:						I/O
	// Parameter:						EventDetectionEnable = FALSE
	MODisp_IO5P							: FB_BACnet_MO_IO5P := (
											iParent									:= fbMNode,
											sDescription							:= '\/Test MO Befehl (IO)',
											sStateText								:= [ 'Aus', 'Stufe 1', 'Stufe 2', 'Stufe 3', 'Stufe 4' ],
											bEventDetectionEnable					:= FALSE
										);
END_VAR
// --- Misc: ---------------------------------------------------------------------------------------------------------------------------------------
VAR_INPUT		
	fbMscNode							: FB_BACnet_View := (
											iParent									:= fbLibNode,
											eNodeType								:= E_BACnet_NodeType.eArea,
											sObjectName								:= '\/Misc',
											sDescription							:= '\/Miscellaneous');
											
	Dev01								: FB_BACnet_Device := (
											iParent									:= fbMscNode,
											sDescription							:= '\/My Device',
											sLocation								:= 'Verl');
											
	LOOP								: FB_BACnet_Loop := (
											iParent									:= fbMscNode,
											sDescription							:= '\/Test Loop',
											eOutputUnit								:= E_BA_Unit.eOther_Percent,
											eAction									:= E_BA_Action.eReverse,
											fPropertionalConstant					:= 5.0,
											fIntegralConstant						:= 180,
											nNotificationClass						:= 10,
											bEventEnable							:= [ FALSE, FALSE, FALSE ],
											sEventMessageTextsConfig				:= [ '\/Überschritten', '\/Fehler', '\/Normal' ]);

	CAL01								: FB_BACnet_Cal := (
											iParent									:= fbMscNode,
											sDescription							:= '\/Kalender 1',
											tDateList := [(
												eType								:= E_BA_DateValChoice.eDate,
												uDate								:= F_BA_DateVal(2020,E_BA_Month.eApril,10)),
											(
												eType								:= E_BA_DateValChoice.eDateRange,
												uDate								:= F_BA_DateRangeVal(nFromYear:=2020,E_BA_Month.eApril,10, nToYear:=2021,E_BA_Month.eMay,11)),
											(
												eType								:= E_BA_DateValChoice.eWeekNDay,
												uDate								:= F_BA_WeekNDayVal(E_BA_Weekday.eFriday, E_BA_Week.eWeek1, E_BA_Month.eFebruary))
											]);
	CAL02								: FB_BACnet_Cal := (
											iParent									:= fbMscNode,
											sDescription							:= '\/Kalender 2');
	CAL03								: FB_BACnet_Cal := (
											iParent									:= fbMscNode,
											sDescription							:= '\/Kalender 3');
	
	// Intention:						Scheduler for analog values
	// Parameter:						tWeek = F_BACnet_SchedWeeklyXxA(...)
	//									tCalendar = [(...), (...), (...)]
	//									tException = [(..., F_BACnet_SchedEntryXxA(...)), (..., F_BACnet_SchedEntryXxA(...)), (..., F_BACnet_SchedEntryXxA(...)), (..., [10:00h > 1.0],[11:00h > null])]
	SchedA								: FB_BACnet_SchedA := (
											iParent									:= fbMscNode,
											sDescription							:= '\/Scheduler Analog',
											tWeek									:= F_BACnet_SchedWeekly3xA(E_BA_Weekday.eMonday, E_BA_Weekday.eFriday, T#0H, 0.0, T#6H, 5.0, T#20H, 0.0),
											tCalendar := [(
												iRefCalendar						:= CAL01,
												stEntry								:= F_BACnet_SchedEntry1xA(T#0H, 2.0)),
											(
												iRefCalendar						:= CAL02,
												stEntry								:= F_BACnet_SchedEntry1xA(T#10H, 3.4)),
											(
												iRefCalendar						:= CAL03,
												stEntry								:= F_BACnet_SchedEntry3xA(T#0H, 5, T#6H, 7, T#20H, 8))
											],
											tException := [(
												eType								:= E_BA_DateValChoice.eDate,
												uDate								:= F_BA_DateVal(2020,E_BA_Month.eApril,10),
												stEntry								:= F_BACnet_SchedEntry1xA(T#0H, 0.0)),
											(
												eType								:= E_BA_DateValChoice.eDateRange,
												uDate								:= F_BA_DateRangeVal(nFromYear:=2020,E_BA_Month.eApril,10, nToYear:=2021,E_BA_Month.eMay,11),
												stEntry								:= F_BACnet_SchedEntry3xA(T#0H, 0.0, T#6H, 5.0, T#20H, 0.0)),
											(
												eType								:= E_BA_DateValChoice.eWeekNDay,
												uDate								:= F_BA_WeekNDayVal(E_BA_Weekday.eFriday, E_BA_Week.eWeek1, E_BA_Month.eFebruary),
												stEntry								:= F_BACnet_SchedEntry3xA(T#0H, 0.0, T#6H, 5.0, T#20H, 0.0)),
											(
												eType								:= E_BA_DateValChoice.eDate,
												uDate								:= F_BA_DateVal(2019,E_BA_Month.eJune,20),
												stEntry := [(
													eState							:= E_BA_SchedEntryState.eValue,
													stTime							:= F_BA_ToSTTime(T#10H),
													uValue							:= F_BA_RVal(1.0)),
												(
													eState							:= E_BA_SchedEntryState.eNull,
													stTime							:= F_BA_ToSTTime(T#11H)
												)]
											)]);
	
	// Intention:						Scheduler for boolean values
	// Parameter:						tWeek = F_BACnet_SchedWeeklyXxB(...)
	//									tCalendar = F_BACnet_SchedCalendar(...)
	SchedB_AssignTestCal2Reference		: BOOL;
	SchedB								: FB_BACnet_SchedB := (
											iParent									:= fbMscNode,
											sDescription							:= '\/Scheduler Bool',
											tWeek									:= F_BACnet_SchedWeekly3xB(E_BA_Weekday.eMonday, E_BA_Weekday.eFriday, T#0H, FALSE, T#6H, TRUE, T#20H, FALSE),
											tCalendar								:= F_BACnet_SchedCalendar(CAL01, 0, 0));
	
	// Intention:						Scheduler for multistate values
	SchedM								: FB_BACnet_SchedM := (
											iParent									:= fbMscNode,
											sDescription							:= '\/Scheduler Multistate',
											tWeek									:= F_BACnet_SchedWeekly3xM(E_BA_Weekday.eMonday, E_BA_Weekday.eFriday, T#0H, 1, T#6H, 2, T#20H, 1));
	
	EventLog_NC11						: FB_BACnet_EventLog := (
											iParent									:= fbMscNode,
											sDescription							:= '\/Event Log für NC11',
											nNotificationClass						:= 11,
											bEventEnable							:= [ TRUE, TRUE, FALSE ],
											sEventMessageTextsConfig				:= [ '\/Überschritten', '\/Fehler', '\/Normal' ],
											nProcessId								:= 20011);
	EventLog_NC12						: FB_BACnet_EventLog := (
											iParent									:= fbMscNode,
											sDescription							:= '\/Event Log für NC12',
											nNotificationClass						:= 11,
											bEventEnable							:= [ TRUE, TRUE, FALSE ],
											sEventMessageTextsConfig				:= [ '\/Überschritten', '\/Fehler', '\/Normal' ],
											nProcessId								:= 20012);

	// (BETA) ... TODO
	// SCHED_Multistate : FB_BACnet_SchedMultistate;
	
	TLog_AssignTestReference			: BOOL;
	TLog_ReadReference					: BOOL;
	TLog_LogReferenceInfo				: BOOL;
	TLog								: FB_BACnet_TLog := (
											iParent									:= fbMscNode,
											sDescription							:= '\/Trend',
											nNotificationClass						:= 11,
											bEventEnable							:= [ TRUE, TRUE, FALSE ],
											sEventMessageTextsConfig				:= [ '\/Überschritten', '\/Fehler', '\/Normal' ],
											stStartTime								:= F_BA_ToSTDateTime(DT#2010-01-01-00:00),
											stDeviceObjPropRef := (
												// ePropertyId						:= PropPresentValue,
												iObject								:= AVSp));
	
	TLogMulti							: FB_BACnet_TLM := (
											iParent									:= fbMscNode,
											sDescription							:= '\/Trend Multiple',
											nNotificationClass						:= 11);
											
	
	fbNCNode							: FB_BA_Server_NC01 := (
											iParent									:= fbMscNode,
											sObjectName								:= '\/NC',
											sDescription							:= '\/Notification Classes'
										);

	(*
	NC01_Standard						: FB_BACnet_NC := (
											iParent									:= fbMscNode,
											nObjectInstance							:= 11,
											nNotificationClass						:= 11,
											sDescription							:= '\/Test NC01 Standard',
											bAckRequired							:= [ TRUE, TRUE, FALSE ],
											nPriority								:= [ 10, 11, 12 ]);
	NC02_Extended						: FB_BACnet_NC := (
											iParent									:= fbMscNode,
											nObjectInstance							:= 10,
											nNotificationClass						:= 10,
											sDescription							:= '\/Test NC02 Extended',
											bAckRequired							:= [ TRUE, TRUE, TRUE ],
											nPriority								:= [ 13, 14, 15 ]);
	*)
	
	{attribute 'hide'}
	_stUnusedCmpData					: ST_BACnet_Destination;
	nCompareRecipient_Index				: UINT										:= 0;
	NC03_RecipientTest					: FB_BACnet_NC := (
											iParent									:= fbMscNode,
											nObjectInstance							:= 244,
											nNotificationClass						:= 244,
											sDescription							:= '\/Test NC03 RecipientTest',
											bAckRequired							:= [ TRUE, TRUE, FALSE ],
											nPriority								:= [ 224, 223, 222 ],
											stRecipientList	:= 
												[
													(
														stValidDays					:= (bSunday:=TRUE, bSaturday:=TRUE, bFriday:=TRUE),
														stFromTime					:= F_BA_ToSTTime(T#0H),
														stToTime					:= F_BA_ToSTTime(T#23H59M59S),
														stRecipient					:= F_BACnet_DeviceRecipient(nDeviceInstance:=5),
														nProcessId					:= 20100,
														bIssueConfirmed				:= FALSE
													),
													(
														stValidDays					:= (bSunday:=TRUE, bSaturday:=TRUE),
														stFromTime					:= F_BA_ToSTTime(T#0H),
														stToTime					:= F_BA_ToSTTime(T#23H59M59S),
														stRecipient					:= F_BACnet_EthernetRecipient(nIPAddress1:=192,168,10,200, nPort:=47808, nNetworkNr:=444),
														nProcessId					:= 30100,
														bIssueConfirmed				:= TRUE
													)
													(* (
														stValidDays					:= (bSunday:=TRUE, bSaturday:=TRUE, bFriday:=TRUE),
														stFromTime					:= F_BA_ToSTTime(T#0H),
														stToTime					:= F_BA_ToSTTime(T#23H59M59S),
														stRecipient := (
															eRecipientChoice		:= E_BACnet_RecipientChoice.eDevice,
															stEntry := (
																tDeviceId			:= 20,
																stNetAddr := (
																	eChoice			:= E_BACnet_AddressChoice.eEthernet,
																	eAddress		:= [ 10, 10, 10, 10, 10, 10, 1, 1 ],
																	nNetworkNr		:= 0))),
														nProcessId					:= 20100,
														bIssueConfirmed				:= FALSE
													) *)
												]
											);
END_VAR
// --- Special: ---------------------------------------------------------------------------------------------------------------------------------------
VAR_INPUT		
	fbSpcNode							: FB_BACnet_View := (
											iParent									:= fbLibNode,
											eNodeType								:= E_BACnet_NodeType.eArea,
											sObjectName								:= '\/Spec',
											sDescription							:= '\/Special');
											
	Acc01								: FB_BACnet_Acc := (
											iParent									:= fbSpcNode,
											sDescription							:= '\/Accumulator');
											
	PC01								: FB_BACnet_PC := (
											iParent									:= fbSpcNode,
											sDescription							:= '\/Pulse Converter');
											
	Prog01								: FB_BACnet_Prog := (
											iParent									:= fbSpcNode,
											sDescription							:= '\/Program');
END_VAR

fbLibNode();
IF (fbLibNode.bUpdateCOV) THEN
	nLibNode_UpdateCount := (nLibNode_UpdateCount+1);
END_IF

// Analog:
fbANode();

AV();
AV5P(bEnSfty := AV5P_TestEnSfty);
AVDsp();
AVSp();
AI_TSenRaw(nRawState:=AI_TSenRaw_State, nRawValue:=AI_TSenRaw_DataIn);
AI_TSenProc(fVal:=AI_TSenProc_Value);
AI_TSenIO();
AIDsp_TSenIO();
AO_CmdRaw(nRawValue=>AO_CmdRaw_Out);
AO_CmdIORaw();
AO_CmdRaw5P(bRawOverridden:=(AO_CmdRaw5P_State<>0), nRawValue=>AO_CmdRaw5P_Out);
AO_CmdIO5P();
AODisp_CmdIO5P();
AO_CmdIO();

// Binary:
fbBNode();

BV();
BV5P();
BVDsp();
BVSp();
BI_DstbRaw(bRawValue:=BI_DstbRaw_In);
BI_DstbIO();
BIDsp_SwiIO();
BO_CmdRaw(bRawValue=>BO_CmdRaw_Out);
BO_CmdIO();
BO_CmdRaw5P(bRawValue=>BO_CmdRaw5P_Out, bEnFeedback:=TRUE, bRawValFeedback:=BO_CmdRaw5P_Feedback, bRawOverridden:=BO_CmdRaw5P_OverrIO);
BO_CmdIO5P();
BODisp_CmdIO5P();

// Multistate:
fbMNode();

MV();
MV5P();
MVDsp();
MVSp();
MI_StateRaw(nRawValue:=MI_StateRaw_In);
MI_StateIO();
MIDsp_Swi_StateRaw(nRawValue:=MIDsp_Swi_StateRaw_In);
MO_CmdRaw(nRawValue=>MO_CmdRaw_Out);
MO_Raw5P(nRawValue=>MO_Raw5P_Out);
MODisp_Raw5P(nRawValue=>MODisp_Raw5P_Out);
MODisp_IO5P();

// Misc:
fbMscNode();

Dev01();

LOOP();
CAL01();
CAL02();
CAL03();
SchedA();
IF (SchedB_AssignTestCal2Reference) THEN
	SchedB_AssignTestCal2Reference := FALSE;
	SchedB.tCalendar[2].iRefCalendar := CAL01;
	SchedB.tCalendar[2].stEntry := F_BACnet_SchedEntry1xB(T#11H, TRUE);
END_IF
SchedB();
SchedM();
EventLog_NC11();
EventLog_NC12();
IF (TLog_AssignTestReference) THEN
	TLog_AssignTestReference := FALSE;
	TLog.stDeviceObjPropRef.iObject := SchedA;
	TLog.DeviceObjectPropertyReference := TLog.stDeviceObjPropRef;
END_IF
IF (TLog_ReadReference) THEN
	TLog_ReadReference := FALSE;
	_hRes := TLog.ReadPropertyReference(E_BACnetPropIdentifier.PropLogDeviceObjectProperty, TLog.stDeviceObjPropRef);
	F_BA_LogMessage1(ADSLOG_MSGTYPE_ERROR, 'DEBUG73', 'Read TLog-Ref: Result=0x%x', F_DINT(_hRes));		
END_IF
IF (TLog_LogReferenceInfo) THEN
	TLog_LogReferenceInfo := FALSE;
	IF (TLog.stDeviceObjPropRef.iObject = 0) THEN
		F_BA_LogMessage(ADSLOG_MSGTYPE_ERROR, 'DEBUG80', 'TLog-Ref: 0');
	ELSE
		tTemp := TLog.stDeviceObjPropRef.iObject.ObjectName;
		F_BA_LogMessage1(ADSLOG_MSGTYPE_ERROR, 'DEBUG83', 'TLog-Ref: %s', F_STRING(tTemp));
	END_IF
END_IF
TLog();
TLogMulti();

fbNCNode();
(*
NC01_Standard();
NC02_Extended();
*)
IF (nCompareRecipient_Index <> 0) THEN
	F_BA_Print('Compare Recipient [Unused]', ADR(_stUnusedCmpData), SIZEOF(ST_BACnet_Destination), TRUE, 64);
	F_BA_Print('Compare Recipient [Index]', ADR(NC03_RecipientTest.stRecipientList[nCompareRecipient_Index]), SIZEOF(ST_BACnet_Destination), TRUE, 64);
	
	nCompareRecipient_Index := TO_UINT(F_BA_GetUsedEntryCount(ADR(NC03_RecipientTest.stRecipientList), 1, BACnet_Param.nNC_RecipientArraySize, _stUnusedCmpData));
	F_BA_LogMessage1(ADSLOG_MSGTYPE_ERROR, 'Compare Recipient', 'Recipient Count: %d', F_UINT(nCompareRecipient_Index));
	
	nCompareRecipient_Index := 0;
END_IF
NC03_RecipientTest();

// Special:
fbSpcNode();

Acc01();
PC01();
Prog01();

END_PROGRAM

// TEST/TestPackage/PERFORMANCE_MIX
PROGRAM PERFORMANCE_MIX
VAR
	i : UDINT;
	bPerf : BOOL := TRUE;
	bOriginal : BOOL := FALSE;
	arrAV   : ARRAY[0..199] OF FB_BACnet_AV;
	arrBV   : ARRAY[0..199] OF FB_BACnet_BV;
	arrMV   : ARRAY[0..199] OF FB_BACnet_MV;
	arrBI   : ARRAY[0..99] OF FB_BACnet_BI_IO;
	arrAI   : ARRAY[0..49] OF FB_BACnet_AI;
	arrAO  	: ARRAY[0..49] OF FB_BACnet_AO_IO;
	arrBO   : ARRAY[0..49] OF FB_BACnet_BO_IO;
	arrMI   : ARRAY[0..49] OF FB_BACnet_MI_IO;
	arrMO   : ARRAY[0..49] OF FB_BACnet_MO_IO;
	arrSCH  : ARRAY[0..19] OF FB_BACnet_SchedB;
	arrTLOG : ARRAY[0..19] OF FB_BACnet_TLog;
	arrCAL  : ARRAY[0..1] OF FB_BACnet_Cal;
	arrNC   : ARRAY[0..4] OF FB_BACnet_NC;
END_VAR

IF bPerf THEN
	FOR i := 0 TO 199 DO
		arrAV[i]( );
		arrBV[i]( );
		arrMV[i]( );
	END_FOR
	
	IF NOT bOriginal THEN
		FOR i := 0 TO 99 DO
			arrBI[i]();
		END_FOR
		
		FOR i := 0 TO 49 DO
			arrAI[i]();
			arrAO[i]();
			arrBO[i]();
			arrMI[i]();
			arrMO[i]();	
		END_FOR
		
		FOR i := 0 TO 19 DO
			arrSCH[i]();
			arrTLOG[i]();
		END_FOR
		
		FOR i := 0 TO 1 DO
			arrCAL[i]();
		END_FOR
		
		FOR i := 0 TO 4 DO
			arrNC[i]();
		END_FOR
	END_IF
END_IF

END_PROGRAM

// TEST/CLIENT_Andreas
PROGRAM CLIENT_Andreas
VAR
	fbClientFb : FB_ClientTest := (Client := (nDeviceInstance := 1));	
	fbClientFb2 : FB_ClientTest := (Client := (nDeviceInstance := 1));	
	
	fbClient : FB_BACnet_Client := (nDeviceInstance := 1, eReadMode:=E_BACnet_CommMode.eRp);
//	fbDevice : FB_BACnetRM_DeviceVisu := (Client:=fbClient);
	fbAo : FB_BACnetRM_AO := (Client:=fbClient, nObjectInstance:=0);
	fbAv : FB_BACnetRM_AV := (Client:=fbClient, nObjectInstance:=0);
	fbBi : FB_BACnetRM_BI := (Client:=fbClient, nObjectInstance:=0);
	
//	fbVisAv0 : FB_BACnetRM_VisuAV := (Client:=fbClient, nObjectInstance:=0);
//	fbVisAv1 : FB_BACnetRM_VisuAV := (Client:=fbClient, nObjectInstance:=1);
//	fbVisAv2 : FB_BACnetRM_VisuAV := (Client:=fbClient, nObjectInstance:=2);
//	fbVisAv3 : FB_BACnetRM_VisuAV := (Client:=fbClient, nObjectInstance:=3);
	
	diag : ST_BACnet_Diagnosis;
	scanRes : ARRAY [0..99] OF ST_BACnetRM_ScanResult;
	syncTime : ST_BA_DateTime;
	
	bDiag : BOOL;
	bScan : BOOL;
	bGet : BOOL;
	bSync : BOOL;
	
	fbClient2 : FB_BACnet_Client := (nDeviceInstance := 546);
END_VAR

fbClientFb();
fbClientFb2();
fbClient();
//fbDevice();
fbAv();
FbAo();
fbBi();
//fbVisAv0();
//fbVisAv1();
//fbVisAv2();
//fbVisAv3();

fbClient2();

IF bDiag THEN
	fbClient.Adapter.GetDiagnosis(ADR(diag));
END_IF

IF bScan THEN	
	fbClient.Adapter.StartScan();
	bScan:=FALSE;
END_IF

IF bGet THEN
	fbClient.Adapter.GetScanResult(ADR(scanRes), 100);
	bGet:=FALSE;
END_IF

IF bSync THEN
	fbClient.Adapter.TimeSync(ADR(syncTime), TRUE);
	bSync:=FALSE;
END_IF

END_PROGRAM

// TEST/MAIN
PROGRAM MAIN
VAR
	wDummy			AT %I*	: WORD;
	
	bKillMe11				: BOOL;
	bKillMe12				: BOOL;
END_VAR
VAR
	bInit					: BOOL := TRUE;
	nCycles					: UDINT;
END_VAR
VAR
	bManualWritePersistent	: BOOL;
	tAutoWritePersistent	: TON						:= (PT := T#20S);
	wPersistentData			: FB_WritePersistentData	:= (PORT:=TwinCAT_SystemInfoVarList._AppInfo.AdsPort, TMOUT:=T#1S, MODE:=E_PersistentMode.SPDM_2PASS);
END_VAR

VAR

	TestView							: FB_BACnet_View := (
											eNodeType								:= E_BACnet_NodeType.eArea,
											sObjectName								:= '\/Tst',
											sDescription							:= '\/Test');
											
	AV1									: FB_BACnet_BV;
	AV2									: FB_BACnet_AV := (
											iParent									:= TestView);

END_VAR

nCycles := (nCycles+1);
IF (bInit) THEN
	bInit := FALSE;
END_IF

tAutoWritePersistent(IN := (NOT tAutoWritePersistent.Q));
IF (bManualWritePersistent) OR (tAutoWritePersistent.Q) THEN
	bManualWritePersistent := FALSE;
	wPersistentData(START:=TRUE);
ELSE
	wPersistentData();
	IF (NOT wPersistentData.BUSY) THEN
		wPersistentData.START:=FALSE;
	END_IF
END_IF



//CLIENT();
//CLIENT_Marco();

//PLANT_DEMO();
//LIB();
//RT();

//FB_MAIN();
//PRG_MAIN();
//MAIN_PRG02();


//PERFORMANCE();


TestView();
AV1();
AV2();

END_PROGRAM
